// Check duration for each phase
positionExtrema := ruckig._profiles[0].positionExtrema();
AssertEquals_LREAL(8.0, positionExtrema.Tmax, 1E-9, message:='Profile[0] Tmax incorrect');
AssertEquals_LREAL(3112.370485074103, positionExtrema.Maximum, 1E-9, message:='Profile[0] maximum incorrect');
AssertEquals_LREAL(0.0, positionExtrema.Tmin, 1E-9, message:='Profile[0] Tmin incorrect');
AssertEquals_LREAL(78.42679297249512, positionExtrema.Minimum, 1E-9, message:='Profile[0] minimum incorrect');

positionExtrema := ruckig._profiles[1].positionExtrema();
AssertEquals_LREAL(0.2183891025126522, positionExtrema.Tmax, 1E-9, message:='Profile[1] Tmax incorrect');
AssertEquals_LREAL(46.54452205781156, positionExtrema.Maximum, 1E-9, message:='Profile[1] maximum incorrect');
AssertEquals_LREAL(8.0, positionExtrema.Tmin, 1E-9, message:='Profile[1] Tmin incorrect');
AssertEquals_LREAL(-9787.213398023361, positionExtrema.Minimum, 1E-9, message:='Profile[1] minimum incorrect');

positionExtrema := ruckig._profiles[2].positionExtrema();
AssertEquals_LREAL(0.0494303119629617, positionExtrema.Tmax, 1E-9, message:='Profile[2] Tmax incorrect');
AssertEquals_LREAL(31.710971182106867, positionExtrema.Maximum, 1E-9, message:='Profile[2] maximum incorrect');
AssertEquals_LREAL(8.0, positionExtrema.Tmin, 1E-9, message:='Profile[2] Tmin incorrect');
AssertEquals_LREAL(-8022.928301920572, positionExtrema.Minimum, 1E-9, message:='Profile[2] minimum incorrect');
   

TEST_FINISHED();
END_METHOD

METHOD Test_Trajectory_VelIntrf_HasMinDuration_HasTargetVelocity_HasTargetAcceleration_22
VAR_INST
  ruckig : Struckig.Ruckig(0.001, 3) := (
  
    ControlInterface := ControlInterfaceType.Velocity,
    Synchronization := SynchronizationType.TimeSync,
    MinDuration := 2.0,
    MaxVelocity := [ 2000.0, 2000.0, 2000.0 ],
    MaxAcceleration := [ 20000.0, 20000.0, 20000.0 ],
    MaxJerk := [ 800000.0, 800000.0, 800000.0 ],
    CurrentPosition := [ -79.7347950117767, 19.391476793099315, 7.245161501695378 ],
    CurrentVelocity := [ 143.04128173279923, -597.5124545779606, -118.71564531017145 ],
    CurrentAcceleration := [ 5642.529309782371, -4265.609648746094, 4828.540937996317 ],
    TargetPosition := [ -68.4590507631062, -68.46147249712232, -71.29488743466081 ],
    TargetVelocity := [ -770.5297588001531, -967.3934412952574, 417.4312367444536 ],
    TargetAcceleration := [ -41.66111920833407, 935.4765738277545, -963.8609114010426 ]
  );
  
  positionExtrema : Struckig.PositionExtremaDesc;
END_VAR
TEST('Trajectory_VelIntrf_HasMinDuration_HasTargetVelocity_HasTargetAcceleration_22');

ruckig();

// Check total duration of profiles
AssertEquals_LREAL(Expected := 2.0, Actual := ruckig.Duration, DELTA := 1E-8, Message := 'Duration incorrect');

// Check minimum duration
AssertEquals_LREAL(Expected := ruckig.MinDuration, Actual := ruckig.Duration, DELTA := 1E-8, Message := 'Minimum duration not equals duration');

// Check duration for each phase
positionExtrema := ruckig._profiles[0].positionExtrema();
AssertEquals_LREAL(0.007638802536377481, positionExtrema.Tmax, 1E-9, message:='Profile[0] Tmax incorrect');
AssertEquals_LREAL(-78.53693764605154, positionExtrema.Maximum, 1E-9, message:='Profile[0] maximum incorrect');
AssertEquals_LREAL(2.0, positionExtrema.Tmin, 1E-9, message:='Profile[0] Tmin incorrect');
AssertEquals_LREAL(-684.0560377921786, positionExtrema.Minimum, 1E-9, message:='Profile[0] minimum incorrect');

positionExtrema := ruckig._profiles[1].positionExtrema();
AssertEquals_LREAL(0.0, positionExtrema.Tmax, 1E-9, message:='Profile[1] Tmax incorrect');
AssertEquals_LREAL(19.391476793099315, positionExtrema.Maximum, 1E-9, message:='Profile[1] maximum incorrect');
AssertEquals_LREAL(2.0, positionExtrema.Tmin, 1E-9, message:='Profile[1] Tmin incorrect');
AssertEquals_LREAL(-3142.7217669332654, positionExtrema.Minimum, 1E-9, message:='Profile[1] minimum incorrect');

positionExtrema := ruckig._profiles[2].positionExtrema();
AssertEquals_LREAL(2.0, positionExtrema.Tmax, 1E-9, message:='Profile[2] Tmax incorrect');
AssertEquals_LREAL(2071.1384078495203, positionExtrema.Maximum, 1E-9, message:='Profile[2] maximum incorrect');
AssertEquals_LREAL(0.02502787930237134, positionExtrema.Tmin, 1E-9, message:='Profile[2] Tmin incorrect');
AssertEquals_LREAL(5.768456383094455, positionExtrema.Minimum, 1E-9, message:='Profile[2] minimum incorrect');
   

TEST_FINISHED();
END_METHOD

METHOD Test_Trajectory_VelIntrf_HasMinDuration_HasTargetVelocity_HasTargetAcceleration_23
VAR_INST
  ruckig : Struckig.Ruckig(0.001, 3) := (
  
    ControlInterface := ControlInterfaceType.Velocity,
    Synchronization := SynchronizationType.TimeSync,
    MinDuration := 4.0,
    MaxVelocity := [ 2000.0, 2000.0, 2000.0 ],
    MaxAcceleration := [ 20000.0, 20000.0, 20000.0 ],
    MaxJerk := [ 800000.0, 800000.0, 800000.0 ],
    CurrentPosition := [ 61.37396011937787, 91.70380359961769, -8.257039659155268 ],
    CurrentVelocity := [ -246.00859628849685, -467.85176399454747, -618.5921990326065 ],
    CurrentAcceleration := [ -4298.249657421169, 4989.7430906178615, -9033.185410088885 ],
    TargetPosition := [ -63.08099775805782, -90.41352080290159, -99.37485926962239 ],
    TargetVelocity := [ -239.3077646725386, 919.245352779569, -397.28894892304845 ],
    TargetAcceleration := [ -291.4115348913673, 23.504752198523192, -795.5915465895694 ]
  );
  
  positionExtrema : Struckig.PositionExtremaDesc;
END_VAR
TEST('Trajectory_VelIntrf_HasMinDuration_HasTargetVelocity_HasTargetAcceleration_23');

ruckig();

// Check total duration of profiles
AssertEquals_LREAL(Expected := 4.0, Actual := ruckig.Duration, DELTA := 1E-8, Message := 'Duration incorrect');

// Check minimum duration
AssertEquals_LREAL(Expected := ruckig.MinDuration, Actual := ruckig.Duration, DELTA := 1E-8, Message := 'Minimum duration not equals duration');

// Check duration for each phase
positionExtrema := ruckig._profiles[0].positionExtrema();
AssertEquals_LREAL(0.0, positionExtrema.Tmax, 1E-9, message:='Profile[0] Tmax incorrect');
AssertEquals_LREAL(61.37396011937787, positionExtrema.Maximum, 1E-9, message:='Profile[0] maximum incorrect');
AssertEquals_LREAL(4.0, positionExtrema.Tmin, 1E-9, message:='Profile[0] Tmin incorrect');
AssertEquals_LREAL(-932.2714554581783, positionExtrema.Minimum, 1E-9, message:='Profile[0] minimum incorrect');

positionExtrema := ruckig._profiles[1].positionExtrema();
AssertEquals_LREAL(4.0, positionExtrema.Tmax, 1E-9, message:='Profile[1] Tmax incorrect');
AssertEquals_LREAL(3356.191464991089, positionExtrema.Maximum, 1E-9, message:='Profile[1] maximum incorrect');
AssertEquals_LREAL(0.10412338784096734, positionExtrema.Tmin, 1E-9, message:='Profile[1] Tmin incorrect');
AssertEquals_LREAL(68.24379604148844, positionExtrema.Minimum, 1E-9, message:='Profile[1] minimum incorrect');

positionExtrema := ruckig._profiles[2].positionExtrema();
AssertEquals_LREAL(0.0, positionExtrema.Tmax, 1E-9, message:='Profile[2] Tmax incorrect');
AssertEquals_LREAL(-8.257039659155268, positionExtrema.Maximum, 1E-9, message:='Profile[2] maximum incorrect');
AssertEquals_LREAL(4.0, positionExtrema.Tmin, 1E-9, message:='Profile[2] Tmin incorrect');
AssertEquals_LREAL(-2142.4383401030323, positionExtrema.Minimum, 1E-9, message:='Profile[2] minimum incorrect');
   

TEST_FINISHED();
END_METHOD

METHOD Test_Trajectory_VelIntrf_HasMinDuration_HasTargetVelocity_HasTargetAcceleration_25
VAR_INST
  ruckig : Struckig.Ruckig(0.001, 3) := (
  
    ControlInterface := ControlInterfaceType.Velocity,
    Synchronization := SynchronizationType.TimeSync,
    MinDuration := 5.0,
    MaxVelocity := [ 2000.0, 2000.0, 2000.0 ],
    MaxAcceleration := [ 20000.0, 20000.0, 20000.0 ],
    MaxJerk := [ 800000.0, 800000.0, 800000.0 ],
    CurrentPosition := [ 99.27158709173054, 51.78630599017913, -82.71240030046118 ],
    CurrentVelocity := [ 617.0096879713556, 556.3356400770322, 654.4714219366203 ],
    CurrentAcceleration := [ 574.9072883020708, 8161.605381343747, 7215.343607485673 ],
    TargetPosition := [ -75.73302485201327, -76.60258111111662, -93.84383456920497 ],
    TargetVelocity := [ -134.5020942775601, 636.5230467842334, -659.8475456020238 ],
    TargetAcceleration := [ -262.53891173287866, -851.053910299499, -307.5361794862756 ]
  );
  
  positionExtrema : Struckig.PositionExtremaDesc;
END_VAR
TEST('Trajectory_VelIntrf_HasMinDuration_HasTargetVelocity_HasTargetAcceleration_25');

ruckig();

// Check total duration of profiles
AssertEquals_LREAL(Expected := 5.0, Actual := ruckig.Duration, DELTA := 1E-8, Message := 'Duration incorrect');

// Check minimum duration
AssertEquals_LREAL(Expected := ruckig.MinDuration, Actual := ruckig.Duration, DELTA := 1E-8, Message := 'Minimum duration not equals duration');

// Check duration for each phase
positionExtrema := ruckig._profiles[0].positionExtrema();
AssertEquals_LREAL(5.0, positionExtrema.Tmax, 1E-9, message:='Profile[0] Tmax incorrect');
AssertEquals_LREAL(2457.793957890017, positionExtrema.Maximum, 1E-9, message:='Profile[0] maximum incorrect');
AssertEquals_LREAL(0.0, positionExtrema.Tmin, 1E-9, message:='Profile[0] Tmin incorrect');
AssertEquals_LREAL(99.27158709173054, positionExtrema.Minimum, 1E-9, message:='Profile[0] minimum incorrect');

positionExtrema := ruckig._profiles[1].positionExtrema();
AssertEquals_LREAL(5.0, positionExtrema.Tmax, 1E-9, message:='Profile[1] Tmax incorrect');
AssertEquals_LREAL(12482.220923700503, positionExtrema.Maximum, 1E-9, message:='Profile[1] maximum incorrect');
AssertEquals_LREAL(0.0, positionExtrema.Tmin, 1E-9, message:='Profile[1] Tmin incorrect');
AssertEquals_LREAL(51.78630599017913, positionExtrema.Minimum, 1E-9, message:='Profile[1] minimum incorrect');

positionExtrema := ruckig._profiles[2].positionExtrema();
AssertEquals_LREAL(5.0, positionExtrema.Tmax, 1E-9, message:='Profile[2] Tmax incorrect');
AssertEquals_LREAL(457.83088712667626, positionExtrema.Maximum, 1E-9, message:='Profile[2] maximum incorrect');
AssertEquals_LREAL(0.0, positionExtrema.Tmin, 1E-9, message:='Profile[2] Tmin incorrect');
AssertEquals_LREAL(-82.71240030046118, positionExtrema.Minimum, 1E-9, message:='Profile[2] minimum incorrect');
   

TEST_FINISHED();
END_METHOD

METHOD Test_Trajectory_VelIntrf_HasMinDuration_HasTargetVelocity_HasTargetAcceleration_26
VAR_INST
  ruckig : Struckig.Ruckig(0.001, 3) := (
  
    ControlInterface := ControlInterfaceType.Velocity,
    Synchronization := SynchronizationType.TimeSync,
    MinDuration := 2.0,
    MaxVelocity := [ 2000.0, 2000.0, 2000.0 ],
    MaxAcceleration := [ 20000.0, 20000.0, 20000.0 ],
    MaxJerk := [ 800000.0, 800000.0, 800000.0 ],
    CurrentPosition := [ 47.83664173753348, -4.090200694219973, 75.62715399288581 ],
    CurrentVelocity := [ -412.71660212910535, -344.97977752529744, -662.3972561668236 ],
    CurrentAcceleration := [ 9700.323608694027, 4925.451680171778, 528.779511900253 ],
    TargetPosition := [ -26.350792724711255, -10.804969468053471, -80.84927076896919 ],
    TargetVelocity := [ -661.2515009925905, -544.0751045990595, 389.8586138148876 ],
    TargetAcceleration := [ -326.74185324603604, 477.02942558038353, -127.6960040536186 ]
  );
  
  positionExtrema : Struckig.PositionExtremaDesc;
END_VAR
TEST('Trajectory_VelIntrf_HasMinDuration_HasTargetVelocity_HasTargetAcceleration_26');

ruckig();

// Check total duration of profiles
AssertEquals_LREAL(Expected := 2.0, Actual := ruckig.Duration, DELTA := 1E-8, Message := 'Duration incorrect');

// Check minimum duration
AssertEquals_LREAL(Expected := ruckig.MinDuration, Actual := ruckig.Duration, DELTA := 1E-8, Message := 'Minimum duration not equals duration');

// Check duration for each phase
positionExtrema := ruckig._profiles[0].positionExtrema();
AssertEquals_LREAL(0.0, positionExtrema.Tmax, 1E-9, message:='Profile[0] Tmax incorrect');
AssertEquals_LREAL(47.83664173753348, positionExtrema.Maximum, 1E-9, message:='Profile[0] maximum incorrect');
AssertEquals_LREAL(2.0, positionExtrema.Tmin, 1E-9, message:='Profile[0] Tmin incorrect');
AssertEquals_LREAL(-965.6623915281051, positionExtrema.Minimum, 1E-9, message:='Profile[0] minimum incorrect');

positionExtrema := ruckig._profiles[1].positionExtrema();
AssertEquals_LREAL(0.0, positionExtrema.Tmax, 1E-9, message:='Profile[1] Tmax incorrect');
AssertEquals_LREAL(-4.090200694219973, positionExtrema.Maximum, 1E-9, message:='Profile[1] maximum incorrect');
AssertEquals_LREAL(2.0, positionExtrema.Tmin, 1E-9, message:='Profile[1] Tmin incorrect');
AssertEquals_LREAL(-877.5597601233831, positionExtrema.Minimum, 1E-9, message:='Profile[1] minimum incorrect');

positionExtrema := ruckig._profiles[2].positionExtrema();
AssertEquals_LREAL(0.0, positionExtrema.Tmax, 1E-9, message:='Profile[2] Tmax incorrect');
AssertEquals_LREAL(75.62715399288581, positionExtrema.Maximum, 1E-9, message:='Profile[2] maximum incorrect');
AssertEquals_LREAL(1.9991825530237812, positionExtrema.Tmin, 1E-9, message:='Profile[2] Tmin incorrect');
AssertEquals_LREAL(-196.96292798248453, positionExtrema.Minimum, 1E-9, message:='Profile[2] minimum incorrect');
   

TEST_FINISHED();
END_METHOD

METHOD Test_Trajectory_VelIntrf_HasMinDuration_HasTargetVelocity_HasTargetAcceleration_33
VAR_INST
  ruckig : Struckig.Ruckig(0.001, 3) := (
  
    ControlInterface := ControlInterfaceType.Velocity,
    Synchronization := SynchronizationType.TimeSync,
    MinDuration := 1.0,
    MaxVelocity := [ 2000.0, 2000.0, 2000.0 ],
    MaxAcceleration := [ 20000.0, 20000.0, 20000.0 ],
    MaxJerk := [ 800000.0, 800000.0, 800000.0 ],
    CurrentPosition := [ -49.2031444482373, -51.45640574706518, 70.88792157601674 ],
    CurrentVelocity := [ -496.32492650532754, -32.672137553484845, 433.6351152131574 ],
    CurrentAcceleration := [ 5796.767034802937, 149.52817879179565, 5479.773632181257 ],
    TargetPosition := [ -60.683308313785076, -77.36542095799315, 35.25281163323578 ],
    TargetVelocity := [ -239.87671609275264, 822.5237555037947, -341.77342454738846 ],
    TargetAcceleration := [ 442.7287565429956, -997.6913770242959, -816.4447449025389 ]
  );
  
  positionExtrema : Struckig.PositionExtremaDesc;
END_VAR
TEST('Trajectory_VelIntrf_HasMinDuration_HasTargetVelocity_HasTargetAcceleration_33');

ruckig();

// Check total duration of profiles
AssertEquals_LREAL(Expected := 1.0, Actual := ruckig.Duration, DELTA := 1E-8, Message := 'Duration incorrect');

// Check minimum duration
AssertEquals_LREAL(Expected := ruckig.MinDuration, Actual := ruckig.Duration, DELTA := 1E-8, Message := 'Minimum duration not equals duration');

// Check duration for each phase
positionExtrema := ruckig._profiles[0].positionExtrema();
AssertEquals_LREAL(0.0, positionExtrema.Tmax, 1E-9, message:='Profile[0] Tmax incorrect');
AssertEquals_LREAL(-49.2031444482373, positionExtrema.Maximum, 1E-9, message:='Profile[0] maximum incorrect');
AssertEquals_LREAL(1.0, positionExtrema.Tmin, 1E-9, message:='Profile[0] Tmin incorrect');
AssertEquals_LREAL(-407.7025966385173, positionExtrema.Minimum, 1E-9, message:='Profile[0] minimum incorrect');

positionExtrema := ruckig._profiles[1].positionExtrema();
AssertEquals_LREAL(1.0, positionExtrema.Tmax, 1E-9, message:='Profile[1] Tmax incorrect');
AssertEquals_LREAL(344.3868574234848, positionExtrema.Maximum, 1E-9, message:='Profile[1] maximum incorrect');
AssertEquals_LREAL(0.000885165723529272, positionExtrema.Tmin, 1E-9, message:='Profile[1] Tmin incorrect');
AssertEquals_LREAL(-51.485174951826146, positionExtrema.Minimum, 1E-9, message:='Profile[1] minimum incorrect');

positionExtrema := ruckig._profiles[2].positionExtrema();
AssertEquals_LREAL(0.9999795141123666, positionExtrema.Tmax, 1E-9, message:='Profile[2] Tmax incorrect');
AssertEquals_LREAL(129.085190687188, positionExtrema.Maximum, 1E-9, message:='Profile[2] maximum incorrect');
AssertEquals_LREAL(0.0, positionExtrema.Tmin, 1E-9, message:='Profile[2] Tmin incorrect');
AssertEquals_LREAL(70.88792157601674, positionExtrema.Minimum, 1E-9, message:='Profile[2] minimum incorrect');
   

TEST_FINISHED();
END_METHOD

METHOD Test_Trajectory_VelIntrf_HasMinDuration_HasTargetVelocity_HasTargetAcceleration_37
VAR_INST
  ruckig : Struckig.Ruckig(0.001, 3) := (
  
    ControlInterface := ControlInterfaceType.Velocity,
    Synchronization := SynchronizationType.TimeSync,
    MinDuration := 2.0,
    MaxVelocity := [ 2000.0, 2000.0, 2000.0 ],
    MaxAcceleration := [ 20000.0, 20000.0, 20000.0 ],
    MaxJerk := [ 800000.0, 800000.0, 800000.0 ],
    CurrentPosition := [ -12.004712599902348, 73.67282675877655, -52.349457595484836 ],
    CurrentVelocity := [ 292.20783385007076, -778.1307817801523, -64.33328614652999 ],
    CurrentAcceleration := [ 245.56834991156393, 4188.319168784961, -3762.4320312456057 ],
    TargetPosition := [ 82.49345668673473, 58.903290717842765, 34.45715254310531 ],
    TargetVelocity := [ -333.20598063149066, 685.2693740134762, 482.0796900333503 ],
    TargetAcceleration := [ 240.05556433564402, -666.6421184257438, -752.3384651343332 ]
  );
  
  positionExtrema : Struckig.PositionExtremaDesc;
END_VAR
TEST('Trajectory_VelIntrf_HasMinDuration_HasTargetVelocity_HasTargetAcceleration_37');

ruckig();

// Check total duration of profiles
AssertEquals_LREAL(Expected := 2.0, Actual := ruckig.Duration, DELTA := 1E-8, Message := 'Duration incorrect');

// Check minimum duration
AssertEquals_LREAL(Expected := ruckig.MinDuration, Actual := ruckig.Duration, DELTA := 1E-8, Message := 'Minimum duration not equals duration');

// Check duration for each phase
positionExtrema := ruckig._profiles[0].positionExtrema();
AssertEquals_LREAL(0.0006980853396357632, positionExtrema.Tmax, 1E-9, message:='Profile[0] Tmax incorrect');
AssertEquals_LREAL(-11.80071211848046, positionExtrema.Maximum, 1E-9, message:='Profile[0] maximum incorrect');
AssertEquals_LREAL(2.0, positionExtrema.Tmin, 1E-9, message:='Profile[0] Tmin incorrect');
AssertEquals_LREAL(-52.999031310760635, positionExtrema.Minimum, 1E-9, message:='Profile[0] minimum incorrect');

positionExtrema := ruckig._profiles[1].positionExtrema();
AssertEquals_LREAL(2.0, positionExtrema.Tmax, 1E-9, message:='Profile[1] Tmax incorrect');
AssertEquals_LREAL(1703.4819483796325, positionExtrema.Maximum, 1E-9, message:='Profile[1] maximum incorrect');
AssertEquals_LREAL(0.207432051719431, positionExtrema.Tmin, 1E-9, message:='Profile[1] Tmin incorrect');
AssertEquals_LREAL(-3.8974776087497673, positionExtrema.Minimum, 1E-9, message:='Profile[1] minimum incorrect');

positionExtrema := ruckig._profiles[2].positionExtrema();
AssertEquals_LREAL(2.0, positionExtrema.Tmax, 1E-9, message:='Profile[2] Tmax incorrect');
AssertEquals_LREAL(355.8717476818793, positionExtrema.Maximum, 1E-9, message:='Profile[2] maximum incorrect');
AssertEquals_LREAL(0.005051342367393055, positionExtrema.Tmin, 1E-9, message:='Profile[2] Tmin incorrect');
AssertEquals_LREAL(-52.70524288915402, positionExtrema.Minimum, 1E-9, message:='Profile[2] minimum incorrect');
   

TEST_FINISHED();
END_METHOD

METHOD Test_Trajectory_VelIntrf_HasMinDuration_HasTargetVelocity_HasTargetAcceleration_40
VAR_INST
  ruckig : Struckig.Ruckig(0.001, 3) := (
  
    ControlInterface := ControlInterfaceType.Velocity,
    Synchronization := SynchronizationType.TimeSync,
    MinDuration := 4.0,
    MaxVelocity := [ 2000.0, 2000.0, 2000.0 ],
    MaxAcceleration := [ 20000.0, 20000.0, 20000.0 ],
    MaxJerk := [ 800000.0, 800000.0, 800000.0 ],
    CurrentPosition := [ -76.42035041184897, -68.81061285502989, 60.15861595713818 ],
    CurrentVelocity := [ 424.8413928919874, 178.96533202855449, 765.6862190691088 ],
    CurrentAcceleration := [ 1338.04438518401, 3559.2301009959247, -1023.1564895528609 ],
    TargetPosition := [ -17.943807189703136, 56.757291906819944, -0.6309720814246589 ],
    TargetVelocity := [ -763.7685723303848, 641.2936977777251, -718.0886986858688 ],
    TargetAcceleration := [ 498.71648374610845, -601.18528422182, -73.467606210815 ]
  );
  
  positionExtrema : Struckig.PositionExtremaDesc;
END_VAR
TEST('Trajectory_VelIntrf_HasMinDuration_HasTargetVelocity_HasTargetAcceleration_40');

ruckig();

// Check total duration of profiles
AssertEquals_LREAL(Expected := 4.0, Actual := ruckig.Duration, DELTA := 1E-8, Message := 'Duration incorrect');

// Check minimum duration
AssertEquals_LREAL(Expected := ruckig.MinDuration, Actual := ruckig.Duration, DELTA := 1E-8, Message := 'Minimum duration not equals duration');

// Check duration for each phase
positionExtrema := ruckig._profiles[0].positionExtrema();
AssertEquals_LREAL(0.0020446425392176273, positionExtrema.Tmax, 1E-9, message:='Profile[0] Tmax incorrect');
AssertEquals_LREAL(-75.5500444389785, positionExtrema.Maximum, 1E-9, message:='Profile[0] maximum incorrect');
AssertEquals_LREAL(4.0, positionExtrema.Tmin, 1E-9, message:='Profile[0] Tmin incorrect');
AssertEquals_LREAL(-751.7240555499565, positionExtrema.Minimum, 1E-9, message:='Profile[0] minimum incorrect');

positionExtrema := ruckig._profiles[1].positionExtrema();
AssertEquals_LREAL(4.0, positionExtrema.Tmax, 1E-9, message:='Profile[1] Tmax incorrect');
AssertEquals_LREAL(5988.6562563663865, positionExtrema.Maximum, 1E-9, message:='Profile[1] maximum incorrect');
AssertEquals_LREAL(0.0, positionExtrema.Tmin, 1E-9, message:='Profile[1] Tmin incorrect');
AssertEquals_LREAL(-68.81061285502989, positionExtrema.Minimum, 1E-9, message:='Profile[1] minimum incorrect');

positionExtrema := ruckig._profiles[2].positionExtrema();
AssertEquals_LREAL(0.897558808059484, positionExtrema.Tmax, 1E-9, message:='Profile[2] Tmax incorrect');
AssertEquals_LREAL(380.9463968009695, positionExtrema.Maximum, 1E-9, message:='Profile[2] maximum incorrect');
AssertEquals_LREAL(4.0, positionExtrema.Tmin, 1E-9, message:='Profile[2] Tmin incorrect');
AssertEquals_LREAL(-1230.5349501304436, positionExtrema.Minimum, 1E-9, message:='Profile[2] minimum incorrect');
   

TEST_FINISHED();
END_METHOD

METHOD Test_Trajectory_VelIntrf_HasMinDuration_HasTargetVelocity_HasTargetAcceleration_9
VAR_INST
  ruckig : Struckig.Ruckig(0.001, 3) := (
  
    ControlInterface := ControlInterfaceType.Velocity,
    Synchronization := SynchronizationType.TimeSync,
    MinDuration := 7.0,
    MaxVelocity := [ 2000.0, 2000.0, 2000.0 ],
    MaxAcceleration := [ 20000.0, 20000.0, 20000.0 ],
    MaxJerk := [ 800000.0, 800000.0, 800000.0 ],
    CurrentPosition := [ 65.33675034249944, 20.471874067999465, 17.7936900678952 ],
    CurrentVelocity := [ 251.51375561632767, -883.355945316876, 592.220566480973 ],
    CurrentAcceleration := [ 9181.774579926536, -9976.3302467699, 2745.115542495065 ],
    TargetPosition := [ -63.4605755257718, 16.3093879856457, -25.6649619333392 ],
    TargetVelocity := [ 614.4494968030804, -34.17434532431503, 533.9879492839282 ],
    TargetAcceleration := [ -792.1476751145624, 673.4644110073796, -240.28714730173158 ]
  );
  
  positionExtrema : Struckig.PositionExtremaDesc;
END_VAR
TEST('Trajectory_VelIntrf_HasMinDuration_HasTargetVelocity_HasTargetAcceleration_9');

ruckig();

// Check total duration of profiles
AssertEquals_LREAL(Expected := 7.0, Actual := ruckig.Duration, DELTA := 1E-8, Message := 'Duration incorrect');

// Check minimum duration
AssertEquals_LREAL(Expected := ruckig.MinDuration, Actual := ruckig.Duration, DELTA := 1E-8, Message := 'Minimum duration not equals duration');

// Check duration for each phase
positionExtrema := ruckig._profiles[0].positionExtrema();
AssertEquals_LREAL(7.0, positionExtrema.Tmax, 1E-9, message:='Profile[0] Tmax incorrect');
AssertEquals_LREAL(21441.07705236427, positionExtrema.Maximum, 1E-9, message:='Profile[0] maximum incorrect');
AssertEquals_LREAL(0.0, positionExtrema.Tmin, 1E-9, message:='Profile[0] Tmin incorrect');
AssertEquals_LREAL(65.33675034249944, positionExtrema.Minimum, 1E-9, message:='Profile[0] minimum incorrect');

positionExtrema := ruckig._profiles[1].positionExtrema();
AssertEquals_LREAL(0.0, positionExtrema.Tmax, 1E-9, message:='Profile[1] Tmax incorrect');
AssertEquals_LREAL(20.471874067999465, positionExtrema.Maximum, 1E-9, message:='Profile[1] maximum incorrect');
AssertEquals_LREAL(7.0, positionExtrema.Tmin, 1E-9, message:='Profile[1] Tmin incorrect');
AssertEquals_LREAL(-15783.474903608412, positionExtrema.Minimum, 1E-9, message:='Profile[1] minimum incorrect');

positionExtrema := ruckig._profiles[2].positionExtrema();
AssertEquals_LREAL(7.0, positionExtrema.Tmax, 1E-9, message:='Profile[2] Tmax incorrect');
AssertEquals_LREAL(9053.9566289456, positionExtrema.Maximum, 1E-9, message:='Profile[2] maximum incorrect');
AssertEquals_LREAL(0.0, positionExtrema.Tmin, 1E-9, message:='Profile[2] Tmin incorrect');
AssertEquals_LREAL(17.7936900678952, positionExtrema.Minimum, 1E-9, message:='Profile[2] minimum incorrect');
   

TEST_FINISHED();
END_METHOD

END_FUNCTION_BLOCK

// ---- POUs/MinDurationTest.TcPOU
FUNCTION_BLOCK MinDurationTest EXTENDS TcUnit.FB_TestSuite

Test_Trajectory_HasMinDuration_HasTargetAcceleration_1();
Test_Trajectory_HasMinDuration_HasTargetAcceleration_2();
Test_Trajectory_HasMinDuration_HasTargetAcceleration_3();
Test_Trajectory_HasMinDuration_HasTargetAcceleration_4();
Test_Trajectory_HasMinDuration_HasTargetVelocity_5();
Test_Trajectory_HasMinDuration_HasTargetAcceleration_6();
Test_Trajectory_HasMinDuration_7();
Test_Trajectory_HasMinDuration_8();
Test_Trajectory_HasMinDuration_HasTargetVelocity_9();
Test_Trajectory_HasMinDuration_HasTargetVelocity_HasTargetAcceleration_10();
Test_Trajectory_HasMinDuration_HasTargetAcceleration_11();
Test_Trajectory_HasMinDuration_HasTargetVelocity_HasTargetAcceleration_12();
Test_Trajectory_HasMinDuration_13();
Test_Trajectory_HasMinDuration_14();
Test_Trajectory_HasMinDuration_HasTargetVelocity_HasTargetAcceleration_15();
Test_Trajectory_HasMinDuration_HasTargetVelocity_16();
Test_Trajectory_HasMinDuration_HasTargetAcceleration_17();
Test_Trajectory_HasMinDuration_HasTargetVelocity_HasTargetAcceleration_18();
Test_Trajectory_HasMinDuration_19();
Test_Trajectory_HasMinDuration_HasTargetVelocity_HasTargetAcceleration_20();

METHOD Test_Trajectory_HasMinDuration_13
VAR_INST
  ruckig : Struckig.Ruckig(0.001, 3) := (
  
    Synchronization := SynchronizationType.TimeSync,
    MinDuration := 8.0,
    MaxVelocity := [ 2000.0, 2000.0, 2000.0 ],
    MaxAcceleration := [ 20000.0, 20000.0, 20000.0 ],
    MaxJerk := [ 800000.0, 800000.0, 800000.0 ],
    CurrentPosition := [ 1.1694773064989192, -79.79875434933777, -86.29153082024368 ],
    CurrentVelocity := [ 876.2379533240828, 909.0293542700074, 204.90724883608482 ],
    CurrentAcceleration := [ -68.09095586171134, 4894.443101566274, 4257.694972396241 ],
    TargetPosition := [ -34.92331212819428, 11.554557728133503, 4.460284190197925 ],
    TargetVelocity := [ 0.0, 0.0, 0.0 ],
    TargetAcceleration := [ 0.0, 0.0, 0.0 ]
  );
  
  positionExtrema : Struckig.PositionExtremaDesc;
END_VAR
TEST('Trajectory_HasMinDuration_13');

ruckig();

// Check total duration of profiles
AssertEquals_LREAL(Expected := 8.0, Actual := ruckig.Duration, DELTA := 1E-8, Message := 'Duration incorrect');

// Check minimum duration
AssertEquals_LREAL(Expected := 8.0, Actual := ruckig.Duration, DELTA := 1E-8, Message := 'Duration incorrect');

// Check duration for each phase
positionExtrema := ruckig._profiles[0].positionExtrema();
AssertEquals_LREAL(0.06457933411638962, positionExtrema.Tmax, 1E-9, message:='Profile[0] Tmax incorrect');
AssertEquals_LREAL(31.162316883962312, positionExtrema.Maximum, 1E-9, message:='Profile[0] maximum incorrect');
AssertEquals_LREAL(7.999999999999999, positionExtrema.Tmin, 1E-9, message:='Profile[0] Tmin incorrect');
AssertEquals_LREAL(-34.92331212819428, positionExtrema.Minimum, 1E-9, message:='Profile[0] minimum incorrect');

positionExtrema := ruckig._profiles[1].positionExtrema();
AssertEquals_LREAL(8.0, positionExtrema.Tmax, 1E-9, message:='Profile[1] Tmax incorrect');
AssertEquals_LREAL(11.554557728133503, positionExtrema.Maximum, 1E-9, message:='Profile[1] maximum incorrect');
AssertEquals_LREAL(0.0, positionExtrema.Tmin, 1E-9, message:='Profile[1] Tmin incorrect');
AssertEquals_LREAL(-79.79875434933777, positionExtrema.Minimum, 1E-9, message:='Profile[1] minimum incorrect');

positionExtrema := ruckig._profiles[2].positionExtrema();
AssertEquals_LREAL(8.0, positionExtrema.Tmax, 1E-9, message:='Profile[2] Tmax incorrect');
AssertEquals_LREAL(4.460284190197925, positionExtrema.Maximum, 1E-9, message:='Profile[2] maximum incorrect');
AssertEquals_LREAL(0.0, positionExtrema.Tmin, 1E-9, message:='Profile[2] Tmin incorrect');
AssertEquals_LREAL(-86.29153082024368, positionExtrema.Minimum, 1E-9, message:='Profile[2] minimum incorrect');
   

TEST_FINISHED();
END_METHOD

METHOD Test_Trajectory_HasMinDuration_14
VAR_INST
  ruckig : Struckig.Ruckig(0.001, 3) := (
  
    Synchronization := SynchronizationType.TimeSync,
    MinDuration := 7.0,
    MaxVelocity := [ 2000.0, 2000.0, 2000.0 ],
    MaxAcceleration := [ 20000.0, 20000.0, 20000.0 ],
    MaxJerk := [ 800000.0, 800000.0, 800000.0 ],
    CurrentPosition := [ 9.590430768397383, 39.54262361303532, 47.91880435556814 ],
    CurrentVelocity := [ -279.73110233883074, -397.2798941946028, -792.783818655297 ],
    CurrentAcceleration := [ 9419.249088701486, -5244.89074121808, -9282.308244489752 ],
    TargetPosition := [ 70.18041902211951, 76.40810294125586, -12.064967166259137 ],
    TargetVelocity := [ 0.0, 0.0, 0.0 ],
    TargetAcceleration := [ 0.0, 0.0, 0.0 ]
  );
  
  positionExtrema : Struckig.PositionExtremaDesc;
END_VAR
TEST('Trajectory_HasMinDuration_14');

ruckig();

// Check total duration of profiles
AssertEquals_LREAL(Expected := 7.0, Actual := ruckig.Duration, DELTA := 1E-8, Message := 'Duration incorrect');

// Check minimum duration
AssertEquals_LREAL(Expected := 7.0, Actual := ruckig.Duration, DELTA := 1E-8, Message := 'Duration incorrect');

// Check duration for each phase
positionExtrema := ruckig._profiles[0].positionExtrema();
AssertEquals_LREAL(7.0, positionExtrema.Tmax, 1E-9, message:='Profile[0] Tmax incorrect');
AssertEquals_LREAL(70.18041902211951, positionExtrema.Maximum, 1E-9, message:='Profile[0] maximum incorrect');
AssertEquals_LREAL(0.024939596648417404, positionExtrema.Tmin, 1E-9, message:='Profile[0] Tmin incorrect');
AssertEquals_LREAL(6.5259576965994945, positionExtrema.Minimum, 1E-9, message:='Profile[0] minimum incorrect');

positionExtrema := ruckig._profiles[1].positionExtrema();
AssertEquals_LREAL(6.999999999999999, positionExtrema.Tmax, 1E-9, message:='Profile[1] Tmax incorrect');
AssertEquals_LREAL(76.40810294125586, positionExtrema.Maximum, 1E-9, message:='Profile[1] maximum incorrect');
AssertEquals_LREAL(0.0482688279337284, positionExtrema.Tmin, 1E-9, message:='Profile[1] Tmin incorrect');
AssertEquals_LREAL(27.490923337843135, positionExtrema.Minimum, 1E-9, message:='Profile[1] minimum incorrect');

positionExtrema := ruckig._profiles[2].positionExtrema();
AssertEquals_LREAL(0.0, positionExtrema.Tmax, 1E-9, message:='Profile[2] Tmax incorrect');
AssertEquals_LREAL(47.91880435556814, positionExtrema.Maximum, 1E-9, message:='Profile[2] maximum incorrect');
AssertEquals_LREAL(7.0, positionExtrema.Tmin, 1E-9, message:='Profile[2] Tmin incorrect');
AssertEquals_LREAL(-12.064967166259137, positionExtrema.Minimum, 1E-9, message:='Profile[2] minimum incorrect');
   

TEST_FINISHED();
END_METHOD

METHOD Test_Trajectory_HasMinDuration_19
VAR_INST
  ruckig : Struckig.Ruckig(0.001, 3) := (
  
    Synchronization := SynchronizationType.TimeSync,
    MinDuration := 3.0,
    MaxVelocity := [ 2000.0, 2000.0, 2000.0 ],
    MaxAcceleration := [ 20000.0, 20000.0, 20000.0 ],
    MaxJerk := [ 800000.0, 800000.0, 800000.0 ],
    CurrentPosition := [ 19.6107174579693, -14.671676826720102, -83.4266917323848 ],
    CurrentVelocity := [ -926.4357934162077, 856.3688940409422, -76.05611387446447 ],
    CurrentAcceleration := [ 8950.685844022108, -6737.3624163819, 7093.876397069776 ],
    TargetPosition := [ 45.75525505687679, -17.630601082354573, 68.42483173219557 ],
    TargetVelocity := [ 0.0, 0.0, 0.0 ],
    TargetAcceleration := [ 0.0, 0.0, 0.0 ]
  );
  
  positionExtrema : Struckig.PositionExtremaDesc;
END_VAR
TEST('Trajectory_HasMinDuration_19');

ruckig();

// Check total duration of profiles
AssertEquals_LREAL(Expected := 3.0, Actual := ruckig.Duration, DELTA := 1E-8, Message := 'Duration incorrect');

// Check minimum duration
AssertEquals_LREAL(Expected := 3.0, Actual := ruckig.Duration, DELTA := 1E-8, Message := 'Duration incorrect');

// Check duration for each phase
positionExtrema := ruckig._profiles[0].positionExtrema();
AssertEquals_LREAL(3.0, positionExtrema.Tmax, 1E-9, message:='Profile[0] Tmax incorrect');
AssertEquals_LREAL(45.75525505687679, positionExtrema.Maximum, 1E-9, message:='Profile[0] maximum incorrect');
AssertEquals_LREAL(0.05690150806828992, positionExtrema.Tmin, 1E-9, message:='Profile[0] Tmin incorrect');
AssertEquals_LREAL(-5.546975088681035, positionExtrema.Minimum, 1E-9, message:='Profile[0] minimum incorrect');

positionExtrema := ruckig._profiles[1].positionExtrema();
AssertEquals_LREAL(0.05654489225740592, positionExtrema.Tmax, 1E-9, message:='Profile[1] Tmax incorrect');
AssertEquals_LREAL(8.500086769282458, positionExtrema.Maximum, 1E-9, message:='Profile[1] maximum incorrect');
AssertEquals_LREAL(2.9999999999999996, positionExtrema.Tmin, 1E-9, message:='Profile[1] Tmin incorrect');
AssertEquals_LREAL(-17.630601082354573, positionExtrema.Minimum, 1E-9, message:='Profile[1] minimum incorrect');

positionExtrema := ruckig._profiles[2].positionExtrema();
AssertEquals_LREAL(3.0, positionExtrema.Tmax, 1E-9, message:='Profile[2] Tmax incorrect');
AssertEquals_LREAL(68.42483173219557, positionExtrema.Maximum, 1E-9, message:='Profile[2] maximum incorrect');
AssertEquals_LREAL(0.007991851854731072, positionExtrema.Tmin, 1E-9, message:='Profile[2] Tmin incorrect');
AssertEquals_LREAL(-83.74565322946518, positionExtrema.Minimum, 1E-9, message:='Profile[2] minimum incorrect');
   

TEST_FINISHED();
END_METHOD

METHOD Test_Trajectory_HasMinDuration_7
VAR_INST
  ruckig : Struckig.Ruckig(0.001, 3) := (
  
    Synchronization := SynchronizationType.TimeSync,
    MinDuration := 3.0,
    MaxVelocity := [ 2000.0, 2000.0, 2000.0 ],
    MaxAcceleration := [ 20000.0, 20000.0, 20000.0 ],
    MaxJerk := [ 800000.0, 800000.0, 800000.0 ],
    CurrentPosition := [ -29.448435809827217, 90.57043249467455, -42.4422398449114 ],
    CurrentVelocity := [ -441.1423852905707, 792.9273075694584, 308.64691156030153 ],
    CurrentAcceleration := [ -114.57718650638526, -7587.445490507809, 1437.7422990266587 ],
    TargetPosition := [ -44.03078989692402, 83.77708613438409, -82.0575436244257 ],
    TargetVelocity := [ 0.0, 0.0, 0.0 ],
    TargetAcceleration := [ 0.0, 0.0, 0.0 ]
  );
  
  positionExtrema : Struckig.PositionExtremaDesc;
END_VAR
TEST('Trajectory_HasMinDuration_7');

ruckig();

// Check total duration of profiles
AssertEquals_LREAL(Expected := 3.0, Actual := ruckig.Duration, DELTA := 1E-8, Message := 'Duration incorrect');

// Check minimum duration
AssertEquals_LREAL(Expected := 3.0, Actual := ruckig.Duration, DELTA := 1E-8, Message := 'Duration incorrect');

// Check duration for each phase
positionExtrema := ruckig._profiles[0].positionExtrema();
AssertEquals_LREAL(0.0, positionExtrema.Tmax, 1E-9, message:='Profile[0] Tmax incorrect');
AssertEquals_LREAL(-29.448435809827217, positionExtrema.Maximum, 1E-9, message:='Profile[0] maximum incorrect');
AssertEquals_LREAL(3.0, positionExtrema.Tmin, 1E-9, message:='Profile[0] Tmin incorrect');
AssertEquals_LREAL(-44.03078989692402, positionExtrema.Minimum, 1E-9, message:='Profile[0] minimum incorrect');

positionExtrema := ruckig._profiles[1].positionExtrema();
AssertEquals_LREAL(0.05266649608484671, positionExtrema.Tmax, 1E-9, message:='Profile[1] Tmax incorrect');
AssertEquals_LREAL(110.27502355296447, positionExtrema.Maximum, 1E-9, message:='Profile[1] maximum incorrect');
AssertEquals_LREAL(3.0, positionExtrema.Tmin, 1E-9, message:='Profile[1] Tmin incorrect');
AssertEquals_LREAL(83.77708613438409, positionExtrema.Minimum, 1E-9, message:='Profile[1] minimum incorrect');

positionExtrema := ruckig._profiles[2].positionExtrema();
AssertEquals_LREAL(0.03589522362162333, positionExtrema.Tmax, 1E-9, message:='Profile[2] Tmax incorrect');
AssertEquals_LREAL(-35.88360266407321, positionExtrema.Maximum, 1E-9, message:='Profile[2] maximum incorrect');
AssertEquals_LREAL(3.0000000000000004, positionExtrema.Tmin, 1E-9, message:='Profile[2] Tmin incorrect');
AssertEquals_LREAL(-82.0575436244257, positionExtrema.Minimum, 1E-9, message:='Profile[2] minimum incorrect');
   

TEST_FINISHED();
END_METHOD

METHOD Test_Trajectory_HasMinDuration_8
VAR_INST
  ruckig : Struckig.Ruckig(0.001, 3) := (
  
    Synchronization := SynchronizationType.TimeSync,
    MinDuration := 7.0,
    MaxVelocity := [ 2000.0, 2000.0, 2000.0 ],
    MaxAcceleration := [ 20000.0, 20000.0, 20000.0 ],
    MaxJerk := [ 800000.0, 800000.0, 800000.0 ],
    CurrentPosition := [ -99.24620189721642, 98.804478840699, -87.42756778236038 ],
    CurrentVelocity := [ -829.4036440965908, 623.2680808978928, 45.75080930558306 ],
    CurrentAcceleration := [ -7246.76941372717, 1502.5540766079612, -230.12493771912523 ],
    TargetPosition := [ -96.24866507944863, -68.29579645255217, 3.1547755930834427 ],
    TargetVelocity := [ 0.0, 0.0, 0.0 ],
    TargetAcceleration := [ 0.0, 0.0, 0.0 ]
  );
  
  positionExtrema : Struckig.PositionExtremaDesc;
END_VAR
TEST('Trajectory_HasMinDuration_8');

ruckig();

// Check total duration of profiles
AssertEquals_LREAL(Expected := 7.0, Actual := ruckig.Duration, DELTA := 1E-8, Message := 'Duration incorrect');

// Check minimum duration
AssertEquals_LREAL(Expected := 7.0, Actual := ruckig.Duration, DELTA := 1E-8, Message := 'Duration incorrect');

// Check duration for each phase
positionExtrema := ruckig._profiles[0].positionExtrema();
AssertEquals_LREAL(6.999999999999999, positionExtrema.Tmax, 1E-9, message:='Profile[0] Tmax incorrect');
AssertEquals_LREAL(-96.24866507944863, positionExtrema.Maximum, 1E-9, message:='Profile[0] maximum incorrect');
AssertEquals_LREAL(0.07365733450421347, positionExtrema.Tmin, 1E-9, message:='Profile[0] Tmin incorrect');
AssertEquals_LREAL(-136.26275842325944, positionExtrema.Minimum, 1E-9, message:='Profile[0] minimum incorrect');

positionExtrema := ruckig._profiles[1].positionExtrema();
AssertEquals_LREAL(0.05127223962572218, positionExtrema.Tmax, 1E-9, message:='Profile[1] Tmax incorrect');
AssertEquals_LREAL(117.33454096897361, positionExtrema.Maximum, 1E-9, message:='Profile[1] maximum incorrect');
AssertEquals_LREAL(7.000000000000001, positionExtrema.Tmin, 1E-9, message:='Profile[1] Tmin incorrect');
AssertEquals_LREAL(-68.29579645255217, positionExtrema.Minimum, 1E-9, message:='Profile[1] minimum incorrect');

positionExtrema := ruckig._profiles[2].positionExtrema();
AssertEquals_LREAL(7.000000000000001, positionExtrema.Tmax, 1E-9, message:='Profile[2] Tmax incorrect');
AssertEquals_LREAL(3.1547755930834427, positionExtrema.Maximum, 1E-9, message:='Profile[2] maximum incorrect');
AssertEquals_LREAL(0.0, positionExtrema.Tmin, 1E-9, message:='Profile[2] Tmin incorrect');
AssertEquals_LREAL(-87.42756778236038, positionExtrema.Minimum, 1E-9, message:='Profile[2] minimum incorrect');
   

TEST_FINISHED();
END_METHOD

METHOD Test_Trajectory_HasMinDuration_HasTargetAcceleration_1
VAR_INST
  ruckig : Struckig.Ruckig(0.001, 3) := (
    Synchronization := SynchronizationType.TimeSync,
    MinDuration := 8.0,
    MaxVelocity := [ 2000.0, 2000.0, 2000.0 ],
    MaxAcceleration := [ 20000.0, 20000.0, 20000.0 ],
    MaxJerk := [ 800000.0, 800000.0, 800000.0 ],
    CurrentPosition := [ -19.81606164381961, 13.781968848302611, 8.093103744301672 ],
    CurrentVelocity := [ 726.8874662814426, 243.71684078988915, 635.9493654202183 ],
    CurrentAcceleration := [ 3652.605974217926, 644.8054101513426, -2503.0584587977 ],
    TargetPosition := [ -37.94747764035489, 31.097009748141545, 51.041074550360605 ],
    TargetVelocity := [ 0.0, 0.0, 0.0 ],
    TargetAcceleration := [ -885.392846257796, -430.70238502743985, -347.6934578997044 ]
  );
  
  positionExtrema : Struckig.PositionExtremaDesc;	
END_VAR
TEST('Trajectory_HasMinDuration_HasTargetAcceleration_1');

ruckig();

// Check total duration of profiles
AssertEquals_LREAL(Expected := 8.0, Actual := ruckig.Duration, DELTA := 1E-8, Message := 'Duration incorrect');

// Check minimum duration
AssertEquals_LREAL(Expected := 8.0, Actual := ruckig.Duration, DELTA := 1E-8, Message := 'Duration incorrect');

// Check duration for each phase
positionExtrema := ruckig._profiles[0].positionExtrema();
AssertEquals_LREAL(0.06287595543262448, positionExtrema.Tmax, 1E-9, message:='Profile[0] Tmax incorrect');
AssertEquals_LREAL(6.175884472766756, positionExtrema.Maximum, 1E-9, message:='Profile[0] maximum incorrect');
AssertEquals_LREAL(7.9977865178843555, positionExtrema.Tmin, 1E-9, message:='Profile[0] Tmin incorrect');
AssertEquals_LREAL(-37.94820063785038, positionExtrema.Minimum, 1E-9, message:='Profile[0] minimum incorrect');

positionExtrema := ruckig._profiles[1].positionExtrema();
AssertEquals_LREAL(7.999999999999999, positionExtrema.Tmax, 1E-9, message:='Profile[1] Tmax incorrect');
AssertEquals_LREAL(31.097009748141545, positionExtrema.Maximum, 1E-9, message:='Profile[1] maximum incorrect');
AssertEquals_LREAL(0.0, positionExtrema.Tmin, 1E-9, message:='Profile[1] Tmin incorrect');
AssertEquals_LREAL(13.781968848302611, positionExtrema.Minimum, 1E-9, message:='Profile[1] minimum incorrect');

positionExtrema := ruckig._profiles[2].positionExtrema();
AssertEquals_LREAL(8.0, positionExtrema.Tmax, 1E-9, message:='Profile[2] Tmax incorrect');
AssertEquals_LREAL(51.041074550360605, positionExtrema.Maximum, 1E-9, message:='Profile[2] maximum incorrect');
AssertEquals_LREAL(0.0, positionExtrema.Tmin, 1E-9, message:='Profile[2] Tmin incorrect');
AssertEquals_LREAL(8.093103744301672, positionExtrema.Minimum, 1E-9, message:='Profile[2] minimum incorrect');
   

TEST_FINISHED();
END_METHOD

METHOD Test_Trajectory_HasMinDuration_HasTargetAcceleration_11
VAR_INST
  ruckig : Struckig.Ruckig(0.001, 3) := (
  
    Synchronization := SynchronizationType.TimeSync,
    MinDuration := 1.0,
    MaxVelocity := [ 2000.0, 2000.0, 2000.0 ],
    MaxAcceleration := [ 20000.0, 20000.0, 20000.0 ],
    MaxJerk := [ 800000.0, 800000.0, 800000.0 ],
    CurrentPosition := [ -7.070165280610553, -80.38372522590178, -46.89812209342119 ],
    CurrentVelocity := [ 839.4919555565891, -203.32957691775698, 521.9568411481566 ],
    CurrentAcceleration := [ 3262.1046041862974, -1428.6156287598897, 5033.848829385297 ],
    TargetPosition := [ 39.58959333241566, -77.56627414027115, -4.797228333391573 ],
    TargetVelocity := [ 0.0, 0.0, 0.0 ],
    TargetAcceleration := [ -610.5754269308525, -729.7372379589295, -407.1344521857434 ]
  );
  
  positionExtrema : Struckig.PositionExtremaDesc;
END_VAR
TEST('Trajectory_HasMinDuration_HasTargetAcceleration_11');

ruckig();

// Check total duration of profiles
AssertEquals_LREAL(Expected := 1.0, Actual := ruckig.Duration, DELTA := 1E-8, Message := 'Duration incorrect');

// Check minimum duration
AssertEquals_LREAL(Expected := 1.0, Actual := ruckig.Duration, DELTA := 1E-8, Message := 'Duration incorrect');

// Check duration for each phase
positionExtrema := ruckig._profiles[0].positionExtrema();
AssertEquals_LREAL(1.0, positionExtrema.Tmax, 1E-9, message:='Profile[0] Tmax incorrect');
AssertEquals_LREAL(39.58959333241566, positionExtrema.Maximum, 1E-9, message:='Profile[0] maximum incorrect');
AssertEquals_LREAL(0.0, positionExtrema.Tmin, 1E-9, message:='Profile[0] Tmin incorrect');
AssertEquals_LREAL(-7.070165280610553, positionExtrema.Minimum, 1E-9, message:='Profile[0] minimum incorrect');

positionExtrema := ruckig._profiles[1].positionExtrema();
AssertEquals_LREAL(1.0, positionExtrema.Tmax, 1E-9, message:='Profile[1] Tmax incorrect');
AssertEquals_LREAL(-77.56627414027115, positionExtrema.Maximum, 1E-9, message:='Profile[1] maximum incorrect');
AssertEquals_LREAL(0.030210863301643, positionExtrema.Tmin, 1E-9, message:='Profile[1] Tmin incorrect');
AssertEquals_LREAL(-83.98327189159232, positionExtrema.Minimum, 1E-9, message:='Profile[1] minimum incorrect');

positionExtrema := ruckig._profiles[2].positionExtrema();
AssertEquals_LREAL(1.0000000000000002, positionExtrema.Tmax, 1E-9, message:='Profile[2] Tmax incorrect');
AssertEquals_LREAL(-4.797228333391573, positionExtrema.Maximum, 1E-9, message:='Profile[2] maximum incorrect');
AssertEquals_LREAL(0.0, positionExtrema.Tmin, 1E-9, message:='Profile[2] Tmin incorrect');
AssertEquals_LREAL(-46.89812209342119, positionExtrema.Minimum, 1E-9, message:='Profile[2] minimum incorrect');
   

TEST_FINISHED();
END_METHOD

METHOD Test_Trajectory_HasMinDuration_HasTargetAcceleration_17
VAR_INST
  ruckig : Struckig.Ruckig(0.001, 3) := (
  
    Synchronization := SynchronizationType.TimeSync,
    MinDuration := 10.0,
    MaxVelocity := [ 2000.0, 2000.0, 2000.0 ],
    MaxAcceleration := [ 20000.0, 20000.0, 20000.0 ],
    MaxJerk := [ 800000.0, 800000.0, 800000.0 ],
    CurrentPosition := [ 41.06103962416182, -31.80504488955978, 63.99589133347962 ],
    CurrentVelocity := [ -749.439069786537, -605.1709178805476, -675.8190572055869 ],
    CurrentAcceleration := [ 4505.221832985957, 2158.0191432223, -7626.549080643861 ],
    TargetPosition := [ -49.277633620043005, -77.94196192090983, 7.643571349353522 ],
    TargetVelocity := [ 0.0, 0.0, 0.0 ],
    TargetAcceleration := [ -613.4884636354268, -619.351295536964, -177.16987102998473 ]
  );
  
  positionExtrema : Struckig.PositionExtremaDesc;
END_VAR
TEST('Trajectory_HasMinDuration_HasTargetAcceleration_17');

ruckig();

// Check total duration of profiles
AssertEquals_LREAL(Expected := 10.0, Actual := ruckig.Duration, DELTA := 1E-8, Message := 'Duration incorrect');

// Check minimum duration
AssertEquals_LREAL(Expected := 10.0, Actual := ruckig.Duration, DELTA := 1E-8, Message := 'Duration incorrect');

// Check duration for each phase
positionExtrema := ruckig._profiles[0].positionExtrema();
AssertEquals_LREAL(0.0, positionExtrema.Tmax, 1E-9, message:='Profile[0] Tmax incorrect');
AssertEquals_LREAL(41.06103962416182, positionExtrema.Maximum, 1E-9, message:='Profile[0] maximum incorrect');
AssertEquals_LREAL(9.998466278840914, positionExtrema.Tmin, 1E-9, message:='Profile[0] Tmin incorrect');
AssertEquals_LREAL(-49.27787413825579, positionExtrema.Minimum, 1E-9, message:='Profile[0] minimum incorrect');

positionExtrema := ruckig._profiles[1].positionExtrema();
AssertEquals_LREAL(0.0, positionExtrema.Tmax, 1E-9, message:='Profile[1] Tmax incorrect');
AssertEquals_LREAL(-31.80504488955978, positionExtrema.Maximum, 1E-9, message:='Profile[1] maximum incorrect');
AssertEquals_LREAL(9.99845162176116, positionExtrema.Tmin, 1E-9, message:='Profile[1] Tmin incorrect');
AssertEquals_LREAL(-77.94220940080136, positionExtrema.Minimum, 1E-9, message:='Profile[1] minimum incorrect');

positionExtrema := ruckig._profiles[2].positionExtrema();
AssertEquals_LREAL(0.0, positionExtrema.Tmax, 1E-9, message:='Profile[2] Tmax incorrect');
AssertEquals_LREAL(63.99589133347962, positionExtrema.Maximum, 1E-9, message:='Profile[2] maximum incorrect');
AssertEquals_LREAL(9.999557075322427, positionExtrema.Tmin, 1E-9, message:='Profile[2] Tmin incorrect');
AssertEquals_LREAL(7.643565556420371, positionExtrema.Minimum, 1E-9, message:='Profile[2] minimum incorrect');
   

TEST_FINISHED();
END_METHOD

METHOD Test_Trajectory_HasMinDuration_HasTargetAcceleration_2
VAR_INST
  ruckig : Struckig.Ruckig(0.001, 3) := (
  
    Synchronization := SynchronizationType.TimeSync,
    MinDuration := 9.0,
    MaxVelocity := [ 2000.0, 2000.0, 2000.0 ],
    MaxAcceleration := [ 20000.0, 20000.0, 20000.0 ],
    MaxJerk := [ 800000.0, 800000.0, 800000.0 ],
    CurrentPosition := [ 66.72445317186691, -7.406214437890085, 70.46458426730621 ],
    CurrentVelocity := [ 342.4260974225069, 430.1494125839465, -220.57495791564202 ],
    CurrentAcceleration := [ -4058.8697131936115, -937.4004804082579, -453.3153688510465 ],
    TargetPosition := [ 81.54050823089204, 50.65362401587811, 41.70097854809535 ],
    TargetVelocity := [ 0.0, 0.0, 0.0 ],
    TargetAcceleration := [ -58.178994858405304, 929.3098774625403, 47.05996186659536 ]
  );
  
  positionExtrema : Struckig.PositionExtremaDesc;
END_VAR
TEST('Trajectory_HasMinDuration_HasTargetAcceleration_2');

ruckig();

// Check total duration of profiles
AssertEquals_LREAL(Expected := 9.0, Actual := ruckig.Duration, DELTA := 1E-8, Message := 'Duration incorrect');

// Check minimum duration
AssertEquals_LREAL(Expected := ruckig.MinDuration, Actual := ruckig.Duration, DELTA := 1E-8, Message := 'Duration incorrect');

// Check duration for each phase
positionExtrema := ruckig._profiles[0].positionExtrema();
AssertEquals_LREAL(8.999999999999998, positionExtrema.Tmax, 1E-9, message:='Profile[0] Tmax incorrect');
AssertEquals_LREAL(81.54050823089204, positionExtrema.Maximum, 1E-9, message:='Profile[0] maximum incorrect');
AssertEquals_LREAL(0.0, positionExtrema.Tmin, 1E-9, message:='Profile[0] Tmin incorrect');
AssertEquals_LREAL(66.72445317186691, positionExtrema.Minimum, 1E-9, message:='Profile[0] minimum incorrect');

positionExtrema := ruckig._profiles[1].positionExtrema();
AssertEquals_LREAL(8.997676725306345, positionExtrema.Tmax, 1E-9, message:='Profile[1] Tmax incorrect');
AssertEquals_LREAL(50.65446002386552, positionExtrema.Maximum, 1E-9, message:='Profile[1] maximum incorrect');
AssertEquals_LREAL(0.0, positionExtrema.Tmin, 1E-9, message:='Profile[1] Tmin incorrect');
AssertEquals_LREAL(-7.406214437890085, positionExtrema.Minimum, 1E-9, message:='Profile[1] minimum incorrect');

positionExtrema := ruckig._profiles[2].positionExtrema();
AssertEquals_LREAL(0.0, positionExtrema.Tmax, 1E-9, message:='Profile[2] Tmax incorrect');
AssertEquals_LREAL(70.46458426730621, positionExtrema.Maximum, 1E-9, message:='Profile[2] maximum incorrect');
AssertEquals_LREAL(9.0, positionExtrema.Tmin, 1E-9, message:='Profile[2] Tmin incorrect');
AssertEquals_LREAL(41.70097854809503, positionExtrema.Minimum, 1E-9, message:='Profile[2] minimum incorrect');
   

TEST_FINISHED();
END_METHOD

METHOD Test_Trajectory_HasMinDuration_HasTargetAcceleration_3
VAR_INST
  ruckig : Struckig.Ruckig(0.001, 3) := (
  
    Synchronization := SynchronizationType.TimeSync,
    MinDuration := 7.0,
    MaxVelocity := [ 2000.0, 2000.0, 2000.0 ],
    MaxAcceleration := [ 20000.0, 20000.0, 20000.0 ],
    MaxJerk := [ 800000.0, 800000.0, 800000.0 ],
    CurrentPosition := [ 92.93281918195305, -37.057893567967405, -56.41888208246879 ],
    CurrentVelocity := [ 919.2036906054796, -544.1333420501469, 731.0755464554313 ],
    CurrentAcceleration := [ -7047.99292674085, 7580.284725007419, -3564.1022106007276 ],
    TargetPosition := [ -46.16949731931599, 10.423824279825439, 25.094577416282803 ],
    TargetVelocity := [ 0.0, 0.0, 0.0 ],
    TargetAcceleration := [ -597.0749810615916, 575.2171643962115, 815.8548576022943 ]
  );
  
  positionExtrema : Struckig.PositionExtremaDesc;
END_VAR
TEST('Trajectory_HasMinDuration_HasTargetAcceleration_3');

ruckig();

// Check total duration of profiles
AssertEquals_LREAL(Expected := 7.0, Actual := ruckig.Duration, DELTA := 1E-8, Message := 'Duration incorrect');

// Check minimum duration
AssertEquals_LREAL(Expected := 7.0, Actual := ruckig.Duration, DELTA := 1E-8, Message := 'Duration incorrect');

// Check duration for each phase
positionExtrema := ruckig._profiles[0].positionExtrema();
AssertEquals_LREAL(0.05717797410396826, positionExtrema.Tmax, 1E-9, message:='Profile[0] Tmax incorrect');
AssertEquals_LREAL(118.91548267627095, positionExtrema.Maximum, 1E-9, message:='Profile[0] maximum incorrect');
AssertEquals_LREAL(6.998507312547345, positionExtrema.Tmin, 1E-9, message:='Profile[0] Tmin incorrect');
AssertEquals_LREAL(-46.169719044685195, positionExtrema.Minimum, 1E-9, message:='Profile[0] minimum incorrect');

positionExtrema := ruckig._profiles[1].positionExtrema();
AssertEquals_LREAL(6.99856195708901, positionExtrema.Tmax, 1E-9, message:='Profile[1] Tmax incorrect');
AssertEquals_LREAL(10.424022534884019, positionExtrema.Maximum, 1E-9, message:='Profile[1] maximum incorrect');
AssertEquals_LREAL(0.0403879580291395, positionExtrema.Tmin, 1E-9, message:='Profile[1] Tmin incorrect');
AssertEquals_LREAL(-47.256877517684565, positionExtrema.Minimum, 1E-9, message:='Profile[1] minimum incorrect');

positionExtrema := ruckig._profiles[2].positionExtrema();
AssertEquals_LREAL(6.997960362855993, positionExtrema.Tmax, 1E-9, message:='Profile[2] Tmax incorrect');
AssertEquals_LREAL(25.095143091923283, positionExtrema.Maximum, 1E-9, message:='Profile[2] maximum incorrect');
AssertEquals_LREAL(0.0, positionExtrema.Tmin, 1E-9, message:='Profile[2] Tmin incorrect');
AssertEquals_LREAL(-56.41888208246879, positionExtrema.Minimum, 1E-9, message:='Profile[2] minimum incorrect');
   

TEST_FINISHED();
END_METHOD

METHOD Test_Trajectory_HasMinDuration_HasTargetAcceleration_4
VAR_INST
  ruckig : Struckig.Ruckig(0.001, 3) := (
  
    Synchronization := SynchronizationType.TimeSync,
    MinDuration := 3.0,
    MaxVelocity := [ 2000.0, 2000.0, 2000.0 ],
    MaxAcceleration := [ 20000.0, 20000.0, 20000.0 ],
    MaxJerk := [ 800000.0, 800000.0, 800000.0 ],
    CurrentPosition := [ -0.660339003647124, -95.83458227326918, -56.22509427236879 ],
    CurrentVelocity := [ -379.1557497186742, 437.2615639977953, 470.58690692947357 ],
    CurrentAcceleration := [ 7762.154315281241, -3727.206686180866, 7593.740905155453 ],
    TargetPosition := [ 84.07152685095582, 75.93155527258662, 84.6954649863176 ],
    TargetVelocity := [ 0.0, 0.0, 0.0 ],
    TargetAcceleration := [ -770.0559965976834, 741.3940743654641, -31.453470585175637 ]
  );
  
  positionExtrema : Struckig.PositionExtremaDesc;
END_VAR
TEST('Trajectory_HasMinDuration_HasTargetAcceleration_4');

ruckig();

// Check total duration of profiles
AssertEquals_LREAL(Expected := 3.0, Actual := ruckig.Duration, DELTA := 1E-8, Message := 'Duration incorrect');

// Check minimum duration
AssertEquals_LREAL(Expected := 3.0, Actual := ruckig.Duration, DELTA := 1E-8, Message := 'Duration incorrect');

// Check duration for each phase
positionExtrema := ruckig._profiles[0].positionExtrema();
AssertEquals_LREAL(2.9999999999999996, positionExtrema.Tmax, 1E-9, message:='Profile[0] Tmax incorrect');
AssertEquals_LREAL(84.07152685095582, positionExtrema.Maximum, 1E-9, message:='Profile[0] maximum incorrect');
AssertEquals_LREAL(0.028865029140955737, positionExtrema.Tmin, 1E-9, message:='Profile[0] Tmin incorrect');
AssertEquals_LREAL(-6.050680420215579, positionExtrema.Minimum, 1E-9, message:='Profile[0] minimum incorrect');

positionExtrema := ruckig._profiles[1].positionExtrema();
AssertEquals_LREAL(2.9981465148140867, positionExtrema.Tmax, 1E-9, message:='Profile[1] Tmax incorrect');
AssertEquals_LREAL(75.93197977102668, positionExtrema.Maximum, 1E-9, message:='Profile[1] maximum incorrect');
AssertEquals_LREAL(0.0, positionExtrema.Tmin, 1E-9, message:='Profile[1] Tmin incorrect');
AssertEquals_LREAL(-95.83458227326918, positionExtrema.Minimum, 1E-9, message:='Profile[1] minimum incorrect');

positionExtrema := ruckig._profiles[2].positionExtrema();
AssertEquals_LREAL(2.9999999999999987, positionExtrema.Tmax, 1E-9, message:='Profile[2] Tmax incorrect');
AssertEquals_LREAL(84.69546498631772, positionExtrema.Maximum, 1E-9, message:='Profile[2] maximum incorrect');
AssertEquals_LREAL(0.0, positionExtrema.Tmin, 1E-9, message:='Profile[2] Tmin incorrect');
AssertEquals_LREAL(-56.22509427236879, positionExtrema.Minimum, 1E-9, message:='Profile[2] minimum incorrect');
   

TEST_FINISHED();
END_METHOD

METHOD Test_Trajectory_HasMinDuration_HasTargetAcceleration_6
VAR_INST
  ruckig : Struckig.Ruckig(0.001, 3) := (
  
    Synchronization := SynchronizationType.TimeSync,
    MinDuration := 10.0,
    MaxVelocity := [ 2000.0, 2000.0, 2000.0 ],
    MaxAcceleration := [ 20000.0, 20000.0, 20000.0 ],
    MaxJerk := [ 800000.0, 800000.0, 800000.0 ],
    CurrentPosition := [ 73.95774355738217, 67.34262397589043, 23.586005113842518 ],
    CurrentVelocity := [ -698.8785963385769, -727.2426189740956, 561.2286861746936 ],
    CurrentAcceleration := [ 5180.079571404243, -9987.23908551058, 8369.828846550932 ],
    TargetPosition := [ 26.101611930284065, -62.69432172088365, -69.25146432081932 ],
    TargetVelocity := [ 0.0, 0.0, 0.0 ],
    TargetAcceleration := [ -131.90971166520217, -629.8496867961894, -805.129073987833 ]
  );
  
  positionExtrema : Struckig.PositionExtremaDesc;
END_VAR
TEST('Trajectory_HasMinDuration_HasTargetAcceleration_6');

ruckig();

// Check total duration of profiles
AssertEquals_LREAL(Expected := 10.0, Actual := ruckig.Duration, DELTA := 1E-8, Message := 'Duration incorrect');

// Check minimum duration
AssertEquals_LREAL(Expected := 10.0, Actual := ruckig.Duration, DELTA := 1E-8, Message := 'Duration incorrect');

// Check duration for each phase
positionExtrema := ruckig._profiles[0].positionExtrema();
AssertEquals_LREAL(0.0, positionExtrema.Tmax, 1E-9, message:='Profile[0] Tmax incorrect');
AssertEquals_LREAL(73.95774355738217, positionExtrema.Maximum, 1E-9, message:='Profile[0] maximum incorrect');
AssertEquals_LREAL(9.999670225720838, positionExtrema.Tmin, 1E-9, message:='Profile[0] Tmin incorrect');
AssertEquals_LREAL(26.101609539396815, positionExtrema.Minimum, 1E-9, message:='Profile[0] minimum incorrect');

positionExtrema := ruckig._profiles[1].positionExtrema();
AssertEquals_LREAL(0.0, positionExtrema.Tmax, 1E-9, message:='Profile[1] Tmax incorrect');
AssertEquals_LREAL(67.34262397589043, positionExtrema.Maximum, 1E-9, message:='Profile[1] maximum incorrect');
AssertEquals_LREAL(9.99842537578301, positionExtrema.Tmin, 1E-9, message:='Profile[1] Tmin incorrect');
AssertEquals_LREAL(-62.69458200011703, positionExtrema.Minimum, 1E-9, message:='Profile[1] minimum incorrect');

positionExtrema := ruckig._profiles[2].positionExtrema();
AssertEquals_LREAL(0.06090028897692612, positionExtrema.Tmax, 1E-9, message:='Profile[2] Tmax incorrect');
AssertEquals_LREAL(46.36974939931049, positionExtrema.Maximum, 1E-9, message:='Profile[2] maximum incorrect');
AssertEquals_LREAL(9.99798717731503, positionExtrema.Tmin, 1E-9, message:='Profile[2] Tmin incorrect');
AssertEquals_LREAL(-69.25200797820925, positionExtrema.Minimum, 1E-9, message:='Profile[2] minimum incorrect');
   

TEST_FINISHED();
END_METHOD

METHOD Test_Trajectory_HasMinDuration_HasTargetVelocity_16
VAR_INST
  ruckig : Struckig.Ruckig(0.001, 3) := (
  
    Synchronization := SynchronizationType.TimeSync,
    MinDuration := 7.0,
    MaxVelocity := [ 2000.0, 2000.0, 2000.0 ],
    MaxAcceleration := [ 20000.0, 20000.0, 20000.0 ],
    MaxJerk := [ 800000.0, 800000.0, 800000.0 ],
    CurrentPosition := [ 7.986268223464748, 30.66263768305589, -71.99998699577253 ],
    CurrentVelocity := [ -536.7319233815753, 166.5896044550318, 426.8037118862651 ],
    CurrentAcceleration := [ -3017.084283791076, -9424.883074091185, -1013.896197334474 ],
    TargetPosition := [ -34.478967783797216, 52.15227078186672, -24.73548276773934 ],
    TargetVelocity := [ -753.4402086481915, 518.6153002230694, -127.83329734668075 ],
    TargetAcceleration := [ 0.0, 0.0, 0.0 ]
  );
  
  positionExtrema : Struckig.PositionExtremaDesc;
END_VAR
TEST('Trajectory_HasMinDuration_HasTargetVelocity_16');

ruckig();

// Check total duration of profiles
AssertEquals_LREAL(Expected := 7.0, Actual := ruckig.Duration, DELTA := 1E-8, Message := 'Duration incorrect');

// Check minimum duration
AssertEquals_LREAL(Expected := 7.0, Actual := ruckig.Duration, DELTA := 1E-8, Message := 'Duration incorrect');

// Check duration for each phase
positionExtrema := ruckig._profiles[0].positionExtrema();
AssertEquals_LREAL(0.0, positionExtrema.Tmax, 1E-9, message:='Profile[0] Tmax incorrect');
AssertEquals_LREAL(7.986268223464748, positionExtrema.Maximum, 1E-9, message:='Profile[0] maximum incorrect');
AssertEquals_LREAL(7.000000000000001, positionExtrema.Tmin, 1E-9, message:='Profile[0] Tmin incorrect');
AssertEquals_LREAL(-34.478967783797216, positionExtrema.Minimum, 1E-9, message:='Profile[0] minimum incorrect');

positionExtrema := ruckig._profiles[1].positionExtrema();
AssertEquals_LREAL(7.000000000000002, positionExtrema.Tmax, 1E-9, message:='Profile[1] Tmax incorrect');
AssertEquals_LREAL(52.15227078186672, positionExtrema.Maximum, 1E-9, message:='Profile[1] maximum incorrect');
AssertEquals_LREAL(0.0, positionExtrema.Tmin, 1E-9, message:='Profile[1] Tmin incorrect');
AssertEquals_LREAL(30.66263768305589, positionExtrema.Minimum, 1E-9, message:='Profile[1] minimum incorrect');

positionExtrema := ruckig._profiles[2].positionExtrema();
AssertEquals_LREAL(6.97793366414829, positionExtrema.Tmax, 1E-9, message:='Profile[2] Tmax incorrect');
AssertEquals_LREAL(-23.14319435212213, positionExtrema.Maximum, 1E-9, message:='Profile[2] maximum incorrect');
AssertEquals_LREAL(0.0, positionExtrema.Tmin, 1E-9, message:='Profile[2] Tmin incorrect');
AssertEquals_LREAL(-71.99998699577253, positionExtrema.Minimum, 1E-9, message:='Profile[2] minimum incorrect');
   

TEST_FINISHED();
END_METHOD

METHOD Test_Trajectory_HasMinDuration_HasTargetVelocity_5
VAR_INST
  ruckig : Struckig.Ruckig(0.001, 3) := (
  
    Synchronization := SynchronizationType.TimeSync,
    MinDuration := 4.0,
    MaxVelocity := [ 2000.0, 2000.0, 2000.0 ],
    MaxAcceleration := [ 20000.0, 20000.0, 20000.0 ],
    MaxJerk := [ 800000.0, 800000.0, 800000.0 ],
    CurrentPosition := [ -3.497413438880301, 31.363081204112206, 63.367720727687384 ],
    CurrentVelocity := [ 866.434234141054, -171.78552231675485, 58.6036663712207 ],
    CurrentAcceleration := [ -6318.744631550888, -7187.849982760071, -3339.305374801589 ],
    TargetPosition := [ 53.47504800393719, 97.23185262639063, -88.75469905530662 ],
    TargetVelocity := [ 726.8020091222686, 210.07958633863836, 83.97764431780661 ],
    TargetAcceleration := [ 0.0, 0.0, 0.0 ]
  );
  
  positionExtrema : Struckig.PositionExtremaDesc;
END_VAR
TEST('Trajectory_HasMinDuration_HasTargetVelocity_5');

ruckig();

// Check total duration of profiles
AssertEquals_LREAL(Expected := 4.0, Actual := ruckig.Duration, DELTA := 1E-8, Message := 'Duration incorrect');

// Check minimum duration
AssertEquals_LREAL(Expected := 4.0, Actual := ruckig.Duration, DELTA := 1E-8, Message := 'Duration incorrect');

// Check duration for each phase
positionExtrema := ruckig._profiles[0].positionExtrema();
AssertEquals_LREAL(4.0, positionExtrema.Tmax, 1E-9, message:='Profile[0] Tmax incorrect');
AssertEquals_LREAL(53.47504800393719, positionExtrema.Maximum, 1E-9, message:='Profile[0] maximum incorrect');
AssertEquals_LREAL(0.0, positionExtrema.Tmin, 1E-9, message:='Profile[0] Tmin incorrect');
AssertEquals_LREAL(-3.497413438880301, positionExtrema.Minimum, 1E-9, message:='Profile[0] minimum incorrect');

positionExtrema := ruckig._profiles[1].positionExtrema();
AssertEquals_LREAL(3.9999999999999996, positionExtrema.Tmax, 1E-9, message:='Profile[1] Tmax incorrect');
AssertEquals_LREAL(97.23185262639063, positionExtrema.Maximum, 1E-9, message:='Profile[1] maximum incorrect');
AssertEquals_LREAL(0.03570009228167893, positionExtrema.Tmin, 1E-9, message:='Profile[1] Tmin incorrect');
AssertEquals_LREAL(26.442768005713322, positionExtrema.Minimum, 1E-9, message:='Profile[1] minimum incorrect');

positionExtrema := ruckig._profiles[2].positionExtrema();
AssertEquals_LREAL(0.00882488089698622, positionExtrema.Tmax, 1E-9, message:='Profile[2] Tmax incorrect');
AssertEquals_LREAL(63.66429252791513, positionExtrema.Maximum, 1E-9, message:='Profile[2] maximum incorrect');
AssertEquals_LREAL(3.98506688402464, positionExtrema.Tmin, 1E-9, message:='Profile[2] Tmin incorrect');
AssertEquals_LREAL(-89.5691863512788, positionExtrema.Minimum, 1E-9, message:='Profile[2] minimum incorrect');
   

TEST_FINISHED();
END_METHOD

METHOD Test_Trajectory_HasMinDuration_HasTargetVelocity_9
VAR_INST
  ruckig : Struckig.Ruckig(0.001, 3) := (
  
    Synchronization := SynchronizationType.TimeSync,
    MinDuration := 7.0,
    MaxVelocity := [ 2000.0, 2000.0, 2000.0 ],
    MaxAcceleration := [ 20000.0, 20000.0, 20000.0 ],
    MaxJerk := [ 800000.0, 800000.0, 800000.0 ],
    CurrentPosition := [ 32.77976315061471, 86.05945833221364, 34.11738301725197 ],
    CurrentVelocity := [ -981.2868512691955, 673.690792063916, -116.7982550185385 ],
    CurrentAcceleration := [ -4108.818774560344, 3339.252734800917, -7298.314365481016 ],
    TargetPosition := [ -55.314233526195245, 80.34443440826854, -61.91751423362351 ],
    TargetVelocity := [ 817.0398878216338, -103.40219473844786, -439.1476692838428 ],
    TargetAcceleration := [ 0.0, 0.0, 0.0 ]
  );
  
  positionExtrema : Struckig.PositionExtremaDesc;
END_VAR
TEST('Trajectory_HasMinDuration_HasTargetVelocity_9');

ruckig();

// Check total duration of profiles
AssertEquals_LREAL(Expected := 7.0, Actual := ruckig.Duration, DELTA := 1E-8, Message := 'Duration incorrect');

// Check minimum duration
AssertEquals_LREAL(Expected := 7.0, Actual := ruckig.Duration, DELTA := 1E-8, Message := 'Duration incorrect');

// Check duration for each phase
positionExtrema := ruckig._profiles[0].positionExtrema();
AssertEquals_LREAL(0.0, positionExtrema.Tmax, 1E-9, message:='Profile[0] Tmax incorrect');
AssertEquals_LREAL(32.77976315061471, positionExtrema.Maximum, 1E-9, message:='Profile[0] maximum incorrect');
AssertEquals_LREAL(6.938765999899139, positionExtrema.Tmin, 1E-9, message:='Profile[0] Tmin incorrect');
AssertEquals_LREAL(-82.11714814813035, positionExtrema.Minimum, 1E-9, message:='Profile[0] minimum incorrect');

positionExtrema := ruckig._profiles[1].positionExtrema();
AssertEquals_LREAL(0.060258152451987596, positionExtrema.Tmax, 1E-9, message:='Profile[1] Tmax incorrect');
AssertEquals_LREAL(108.93997970698679, positionExtrema.Maximum, 1E-9, message:='Profile[1] maximum incorrect');
AssertEquals_LREAL(7.0, positionExtrema.Tmin, 1E-9, message:='Profile[1] Tmin incorrect');
AssertEquals_LREAL(80.34443440826854, positionExtrema.Minimum, 1E-9, message:='Profile[1] minimum incorrect');

positionExtrema := ruckig._profiles[2].positionExtrema();
AssertEquals_LREAL(0.0, positionExtrema.Tmax, 1E-9, message:='Profile[2] Tmax incorrect');
AssertEquals_LREAL(34.11738301725197, positionExtrema.Maximum, 1E-9, message:='Profile[2] maximum incorrect');
AssertEquals_LREAL(7.0, positionExtrema.Tmin, 1E-9, message:='Profile[2] Tmin incorrect');
AssertEquals_LREAL(-61.91751423362351, positionExtrema.Minimum, 1E-9, message:='Profile[2] minimum incorrect');
   

TEST_FINISHED();
END_METHOD

METHOD Test_Trajectory_HasMinDuration_HasTargetVelocity_HasTargetAcceleration_10
VAR_INST
  ruckig : Struckig.Ruckig(0.001, 3) := (
  
    Synchronization := SynchronizationType.TimeSync,
    MinDuration := 5.0,
    MaxVelocity := [ 2000.0, 2000.0, 2000.0 ],
    MaxAcceleration := [ 20000.0, 20000.0, 20000.0 ],
    MaxJerk := [ 800000.0, 800000.0, 800000.0 ],
    CurrentPosition := [ -63.70257714146867, 22.730031520740937, -51.56243568859453 ],
    CurrentVelocity := [ -520.8565160201103, 365.56449403589454, 835.823452928573 ],
    CurrentAcceleration := [ 9598.328373658613, -2893.4545241775922, 121.46690068480166 ],
    TargetPosition := [ 22.750797061424464, 74.13128623236747, 69.96760822932885 ],
    TargetVelocity := [ -174.7936793360849, -636.488954459087, -938.8757724326924 ],
    TargetAcceleration := [ 391.8907382899415, -699.6872603922127, 978.1856283310506 ]
  );
  
  positionExtrema : Struckig.PositionExtremaDesc;
END_VAR
TEST('Trajectory_HasMinDuration_HasTargetVelocity_HasTargetAcceleration_10');

ruckig();

// Check total duration of profiles
AssertEquals_LREAL(Expected := 5.0, Actual := ruckig.Duration, DELTA := 1E-8, Message := 'Duration incorrect');

// Check minimum duration
AssertEquals_LREAL(Expected := 5.0, Actual := ruckig.Duration, DELTA := 1E-8, Message := 'Duration incorrect');

// Check duration for each phase
positionExtrema := ruckig._profiles[0].positionExtrema();
AssertEquals_LREAL(4.975346883096284, positionExtrema.Tmax, 1E-9, message:='Profile[0] Tmax incorrect');
AssertEquals_LREAL(25.348702524320338, positionExtrema.Maximum, 1E-9, message:='Profile[0] maximum incorrect');
AssertEquals_LREAL(0.0358766442937755, positionExtrema.Tmin, 1E-9, message:='Profile[0] Tmin incorrect');
AssertEquals_LREAL(-72.4234881857976, positionExtrema.Minimum, 1E-9, message:='Profile[0] minimum incorrect');

positionExtrema := ruckig._profiles[1].positionExtrema();
AssertEquals_LREAL(4.949024471203024, positionExtrema.Tmax, 1E-9, message:='Profile[1] Tmax incorrect');
AssertEquals_LREAL(91.55742573849955, positionExtrema.Maximum, 1E-9, message:='Profile[1] maximum incorrect');
AssertEquals_LREAL(0.0, positionExtrema.Tmin, 1E-9, message:='Profile[1] Tmin incorrect');
AssertEquals_LREAL(22.730031520740937, positionExtrema.Minimum, 1E-9, message:='Profile[1] minimum incorrect');

positionExtrema := ruckig._profiles[2].positionExtrema();
AssertEquals_LREAL(4.933596685985829, positionExtrema.Tmax, 1E-9, message:='Profile[2] Tmax incorrect');
AssertEquals_LREAL(104.72094552143355, positionExtrema.Maximum, 1E-9, message:='Profile[2] maximum incorrect');
AssertEquals_LREAL(0.0, positionExtrema.Tmin, 1E-9, message:='Profile[2] Tmin incorrect');
AssertEquals_LREAL(-51.56243568859453, positionExtrema.Minimum, 1E-9, message:='Profile[2] minimum incorrect');
   

TEST_FINISHED();
END_METHOD

METHOD Test_Trajectory_HasMinDuration_HasTargetVelocity_HasTargetAcceleration_12
VAR_INST
  ruckig : Struckig.Ruckig(0.001, 3) := (
  
    Synchronization := SynchronizationType.TimeSync,
    MinDuration := 8.0,
    MaxVelocity := [ 2000.0, 2000.0, 2000.0 ],
    MaxAcceleration := [ 20000.0, 20000.0, 20000.0 ],
    MaxJerk := [ 800000.0, 800000.0, 800000.0 ],
    CurrentPosition := [ 34.32407664987838, -19.61426768221135, 0.08400152186804632 ],
    CurrentVelocity := [ -637.0909066222588, -315.93942928026286, -768.0946853095916 ],
    CurrentAcceleration := [ 5239.657334131169, -3857.903449466051, 5261.930344314516 ],
    TargetPosition := [ -0.6332298839860186, 7.05929814872006, 84.95032201129774 ],
    TargetVelocity := [ -688.3030057720259, 935.2283186121415, -773.3660434214753 ],
    TargetAcceleration := [ 75.12349151093213, -861.2904239623496, 251.41067093552897 ]
  );
  
  positionExtrema : Struckig.PositionExtremaDesc;
END_VAR
TEST('Trajectory_HasMinDuration_HasTargetVelocity_HasTargetAcceleration_12');

ruckig();

// Check total duration of profiles
AssertEquals_LREAL(Expected := 8.0, Actual := ruckig.Duration, DELTA := 1E-8, Message := 'Duration incorrect');

// Check minimum duration
AssertEquals_LREAL(Expected := 8.0, Actual := ruckig.Duration, DELTA := 1E-8, Message := 'Duration incorrect');

// Check duration for each phase
positionExtrema := ruckig._profiles[0].positionExtrema();
AssertEquals_LREAL(0.0, positionExtrema.Tmax, 1E-9, message:='Profile[0] Tmax incorrect');
AssertEquals_LREAL(34.32407664987838, positionExtrema.Maximum, 1E-9, message:='Profile[0] maximum incorrect');
AssertEquals_LREAL(8.0, positionExtrema.Tmin, 1E-9, message:='Profile[0] Tmin incorrect');
AssertEquals_LREAL(-0.6332298839860186, positionExtrema.Minimum, 1E-9, message:='Profile[0] minimum incorrect');

positionExtrema := ruckig._profiles[1].positionExtrema();
AssertEquals_LREAL(8.0, positionExtrema.Tmax, 1E-9, message:='Profile[1] Tmax incorrect');
AssertEquals_LREAL(7.05929814872006, positionExtrema.Maximum, 1E-9, message:='Profile[1] maximum incorrect');
AssertEquals_LREAL(0.04490272145795441, positionExtrema.Tmin, 1E-9, message:='Profile[1] Tmin incorrect');
AssertEquals_LREAL(-27.725399337897105, positionExtrema.Minimum, 1E-9, message:='Profile[1] minimum incorrect');

positionExtrema := ruckig._profiles[2].positionExtrema();
AssertEquals_LREAL(7.941603003365496, positionExtrema.Tmax, 1E-9, message:='Profile[2] Tmax incorrect');
AssertEquals_LREAL(109.67291667846435, positionExtrema.Maximum, 1E-9, message:='Profile[2] maximum incorrect');
AssertEquals_LREAL(0.05210502444806486, positionExtrema.Tmin, 1E-9, message:='Profile[2] Tmin incorrect');
AssertEquals_LREAL(-19.88492411775111, positionExtrema.Minimum, 1E-9, message:='Profile[2] minimum incorrect');
   

TEST_FINISHED();
END_METHOD

METHOD Test_Trajectory_HasMinDuration_HasTargetVelocity_HasTargetAcceleration_15
VAR_INST
  ruckig : Struckig.Ruckig(0.001, 3) := (
  
    Synchronization := SynchronizationType.TimeSync,
    MinDuration := 6.0,
    MaxVelocity := [ 2000.0, 2000.0, 2000.0 ],
    MaxAcceleration := [ 20000.0, 20000.0, 20000.0 ],
    MaxJerk := [ 800000.0, 800000.0, 800000.0 ],
    CurrentPosition := [ 80.29599725108966, -16.595240167642288, -10.563218674718456 ],
    CurrentVelocity := [ -665.2939916748119, -252.31162160327165, 910.7605496896838 ],
    CurrentAcceleration := [ -6038.086221066726, 5702.712022046548, -5391.38537360544 ],
    TargetPosition := [ -15.947396233027035, -52.93402548041466, -99.24861248238838 ],
    TargetVelocity := [ -82.3068299752083, 810.5242632500622, -475.5452525569576 ],
    TargetAcceleration := [ 797.6779209006231, 304.9451091028675, 294.8876599912337 ]
  );
  
  positionExtrema : Struckig.PositionExtremaDesc;
END_VAR
TEST('Trajectory_HasMinDuration_HasTargetVelocity_HasTargetAcceleration_15');

ruckig();

// Check total duration of profiles
AssertEquals_LREAL(Expected := 6.0, Actual := ruckig.Duration, DELTA := 1E-8, Message := 'Duration incorrect');

// Check minimum duration
AssertEquals_LREAL(Expected := 6.0, Actual := ruckig.Duration, DELTA := 1E-8, Message := 'Duration incorrect');

// Check duration for each phase
positionExtrema := ruckig._profiles[0].positionExtrema();
AssertEquals_LREAL(0.0, positionExtrema.Tmax, 1E-9, message:='Profile[0] Tmax incorrect');
AssertEquals_LREAL(80.29599725108966, positionExtrema.Maximum, 1E-9, message:='Profile[0] maximum incorrect');
AssertEquals_LREAL(5.999999999999999, positionExtrema.Tmin, 1E-9, message:='Profile[0] Tmin incorrect');
AssertEquals_LREAL(-15.947396233027035, positionExtrema.Minimum, 1E-9, message:='Profile[0] minimum incorrect');

positionExtrema := ruckig._profiles[1].positionExtrema();
AssertEquals_LREAL(0.0, positionExtrema.Tmax, 1E-9, message:='Profile[1] Tmax incorrect');
AssertEquals_LREAL(-16.595240167642288, positionExtrema.Maximum, 1E-9, message:='Profile[1] maximum incorrect');
AssertEquals_LREAL(5.939358209422553, positionExtrema.Tmin, 1E-9, message:='Profile[1] Tmin incorrect');
AssertEquals_LREAL(-79.08901602854112, positionExtrema.Minimum, 1E-9, message:='Profile[1] minimum incorrect');

positionExtrema := ruckig._profiles[2].positionExtrema();
AssertEquals_LREAL(0.058957419609001596, positionExtrema.Tmax, 1E-9, message:='Profile[2] Tmax incorrect');
AssertEquals_LREAL(16.2518405159937, positionExtrema.Maximum, 1E-9, message:='Profile[2] maximum incorrect');
AssertEquals_LREAL(6.0, positionExtrema.Tmin, 1E-9, message:='Profile[2] Tmin incorrect');
AssertEquals_LREAL(-99.24861248238838, positionExtrema.Minimum, 1E-9, message:='Profile[2] minimum incorrect');
   

TEST_FINISHED();
END_METHOD

METHOD Test_Trajectory_HasMinDuration_HasTargetVelocity_HasTargetAcceleration_18
VAR_INST
  ruckig : Struckig.Ruckig(0.001, 3) := (
  
    Synchronization := SynchronizationType.TimeSync,
    MinDuration := 6.0,
    MaxVelocity := [ 2000.0, 2000.0, 2000.0 ],
    MaxAcceleration := [ 20000.0, 20000.0, 20000.0 ],
    MaxJerk := [ 800000.0, 800000.0, 800000.0 ],
    CurrentPosition := [ 81.8189456654396, -34.648960679925025, -51.77657021421829 ],
    CurrentVelocity := [ 52.71918271967047, -512.6427429671598, 347.52161587573437 ],
    CurrentAcceleration := [ -463.2079718295354, -9185.891702573537, 7766.274147421525 ],
    TargetPosition := [ 28.57172398615708, 23.600629576782865, -2.4216248210818776 ],
    TargetVelocity := [ 159.80128500214232, -165.6494233580952, 407.13274543851867 ],
    TargetAcceleration := [ -496.57312685360756, 646.2561464861296, 884.0412488799539 ]
  );
  
  positionExtrema : Struckig.PositionExtremaDesc;
END_VAR
TEST('Trajectory_HasMinDuration_HasTargetVelocity_HasTargetAcceleration_18');

ruckig();

// Check total duration of profiles
AssertEquals_LREAL(Expected := 6.0, Actual := ruckig.Duration, DELTA := 1E-8, Message := 'Duration incorrect');

// Check minimum duration
AssertEquals_LREAL(Expected := 6.0, Actual := ruckig.Duration, DELTA := 1E-8, Message := 'Duration incorrect');

// Check duration for each phase
positionExtrema := ruckig._profiles[0].positionExtrema();
AssertEquals_LREAL(0.012217427498857257, positionExtrema.Tmax, 1E-9, message:='Profile[0] Tmax incorrect');
AssertEquals_LREAL(82.2020759262068, positionExtrema.Maximum, 1E-9, message:='Profile[0] maximum incorrect');
AssertEquals_LREAL(5.975125497966807, positionExtrema.Tmin, 1E-9, message:='Profile[0] Tmin incorrect');
AssertEquals_LREAL(26.251513510769477, positionExtrema.Minimum, 1E-9, message:='Profile[0] minimum incorrect');

positionExtrema := ruckig._profiles[1].positionExtrema();
AssertEquals_LREAL(5.9750978983936935, positionExtrema.Tmax, 1E-9, message:='Profile[1] Tmax incorrect');
AssertEquals_LREAL(26.068274316521368, positionExtrema.Maximum, 1E-9, message:='Profile[1] maximum incorrect');
AssertEquals_LREAL(0.059557771163129256, positionExtrema.Tmin, 1E-9, message:='Profile[1] Tmin incorrect');
AssertEquals_LREAL(-55.87398334808502, positionExtrema.Minimum, 1E-9, message:='Profile[1] minimum incorrect');

positionExtrema := ruckig._profiles[2].positionExtrema();
AssertEquals_LREAL(6.0, positionExtrema.Tmax, 1E-9, message:='Profile[2] Tmax incorrect');
AssertEquals_LREAL(-2.4216248210818776, positionExtrema.Maximum, 1E-9, message:='Profile[2] maximum incorrect');
AssertEquals_LREAL(0.0, positionExtrema.Tmin, 1E-9, message:='Profile[2] Tmin incorrect');
AssertEquals_LREAL(-51.77657021421829, positionExtrema.Minimum, 1E-9, message:='Profile[2] minimum incorrect');
   

TEST_FINISHED();
END_METHOD

METHOD Test_Trajectory_HasMinDuration_HasTargetVelocity_HasTargetAcceleration_20
VAR_INST
  ruckig : Struckig.Ruckig(0.001, 3) := (
  
    Synchronization := SynchronizationType.TimeSync,
    MinDuration := 1.0,
    MaxVelocity := [ 2000.0, 2000.0, 2000.0 ],
    MaxAcceleration := [ 20000.0, 20000.0, 20000.0 ],
    MaxJerk := [ 800000.0, 800000.0, 800000.0 ],
    CurrentPosition := [ 74.13037097871606, 50.87684992213954, -35.461969837009065 ],
    CurrentVelocity := [ -104.6717721730954, 978.8741284865525, 932.4293320305519 ],
    CurrentAcceleration := [ -1484.1311843071398, -3303.1671799903806, -254.44992328560875 ],
    TargetPosition := [ -53.87981386222778, -79.63304774882201, 29.944494194232874 ],
    TargetVelocity := [ -444.5052876664206, 76.57672906373682, 439.3701152281369 ],
    TargetAcceleration := [ 223.1822145745084, 144.20762241820466, 871.7177536324762 ]
  );
  
  positionExtrema : Struckig.PositionExtremaDesc;
END_VAR
TEST('Trajectory_HasMinDuration_HasTargetVelocity_HasTargetAcceleration_20');

ruckig();

// Check total duration of profiles
AssertEquals_LREAL(Expected := 1.0, Actual := ruckig.Duration, DELTA := 1E-8, Message := 'Duration incorrect');

// Check minimum duration
AssertEquals_LREAL(Expected := 1.0, Actual := ruckig.Duration, DELTA := 1E-8, Message := 'Duration incorrect');

// Check duration for each phase
positionExtrema := ruckig._profiles[0].positionExtrema();
AssertEquals_LREAL(0.0, positionExtrema.Tmax, 1E-9, message:='Profile[0] Tmax incorrect');
AssertEquals_LREAL(74.13037097871606, positionExtrema.Maximum, 1E-9, message:='Profile[0] maximum incorrect');
AssertEquals_LREAL(1.0, positionExtrema.Tmin, 1E-9, message:='Profile[0] Tmin incorrect');
AssertEquals_LREAL(-53.87981386222778, positionExtrema.Minimum, 1E-9, message:='Profile[0] minimum incorrect');

positionExtrema := ruckig._profiles[1].positionExtrema();
AssertEquals_LREAL(0.05795449228928962, positionExtrema.Tmax, 1E-9, message:='Profile[1] Tmax incorrect');
AssertEquals_LREAL(82.91327789055885, positionExtrema.Maximum, 1E-9, message:='Profile[1] maximum incorrect');
AssertEquals_LREAL(0.9863428350510189, positionExtrema.Tmin, 1E-9, message:='Profile[1] Tmin incorrect');
AssertEquals_LREAL(-80.32577887227478, positionExtrema.Minimum, 1E-9, message:='Profile[1] minimum incorrect');

positionExtrema := ruckig._profiles[2].positionExtrema();
AssertEquals_LREAL(1.0, positionExtrema.Tmax, 1E-9, message:='Profile[2] Tmax incorrect');
AssertEquals_LREAL(29.944494194232874, positionExtrema.Maximum, 1E-9, message:='Profile[2] maximum incorrect');
AssertEquals_LREAL(0.0, positionExtrema.Tmin, 1E-9, message:='Profile[2] Tmin incorrect');
AssertEquals_LREAL(-35.461969837009065, positionExtrema.Minimum, 1E-9, message:='Profile[2] minimum incorrect');
   

TEST_FINISHED();
END_METHOD

END_FUNCTION_BLOCK

// ---- POUs/TargetPosTest.TcPOU
FUNCTION_BLOCK TargetPosTest EXTENDS TcUnit.FB_TestSuite
VAR
  ruckig : Struckig.Ruckig(0.001, 3) := (
  
    Synchronization := SynchronizationType.TimeSync,        
    MaxVelocity := [ 2000.00000000000000000000, 2000.00000000000000000000, 2000.00000000000000000000 ],
    MaxAcceleration := [ 20000.00000000000000000000, 20000.00000000000000000000, 20000.00000000000000000000 ],
    MaxJerk := [ 800000.00000000000000000000, 800000.00000000000000000000, 800000.00000000000000000000 ],
    CurrentPosition := [ 48.86656216713086564596, 31.55963588984187140341, -13.09422790776093847853 ],
    CurrentVelocity := [ -274.21841080128081102885, -440.94461360926254656079, -764.75678162210920163488 ],
    CurrentAcceleration := [ -1478.09700836416959646158, 686.79611869591644790489, -9263.72976579731221136171 ],
    TargetPosition := [ 25.57994474955607699940, -15.83091418217283319336, -38.97164514571973370494 ],
    TargetVelocity := [ 0.00000000000000000000, 0.00000000000000000000, 0.00000000000000000000 ],
    TargetAcceleration := [ 0.00000000000000000000, 0.00000000000000000000, 0.00000000000000000000 ]
  );
  
  positionExtrema : Struckig.PositionExtremaDesc;  
END_VAR

Test_Trajectory_2();;
Test_Trajectory_5();
Test_Trajectory_6();
Test_Trajectory_7();
Test_Trajectory_12();
Test_Trajectory_16(); // this test required to do a more precise implementation of cbrt
Test_Trajectory_30();
Test_Trajectory_32();
Test_Trajectory_33();
Test_Trajectory_40();
Test_Trajectory_49();
Test_Trajectory_53();
Test_Trajectory_59();
Test_Trajectory_62();
Test_Trajectory_64();
Test_Trajectory_65();
Test_Trajectory_68();

METHOD Test_Trajectory_12
VAR_INST
  ruckig : Struckig.Ruckig(0.001, 3) := (
  
    Synchronization := SynchronizationType.TimeSync,        
    MaxVelocity := [ 2000.00000000000000000000, 2000.00000000000000000000, 2000.00000000000000000000 ],
    MaxAcceleration := [ 20000.00000000000000000000, 20000.00000000000000000000, 20000.00000000000000000000 ],
    MaxJerk := [ 800000.00000000000000000000, 800000.00000000000000000000, 800000.00000000000000000000 ],
    CurrentPosition := [ 12.15863849634686744139, 83.56438022017914590833, -29.82534868849941744884 ],
    CurrentVelocity := [ -881.54677264260010360886, -40.22247547933807254594, 795.30816871835008896596 ],
    CurrentAcceleration := [ 6802.73049394882036722265, -2844.95338607063877134351, -3652.21806306270900677191 ],
    TargetPosition := [ 61.24855302996508044089, -54.65891429617437324850, 65.64407005892678625969 ],
    TargetVelocity := [ 0.00000000000000000000, 0.00000000000000000000, 0.00000000000000000000 ],
    TargetAcceleration := [ 0.00000000000000000000, 0.00000000000000000000, 0.00000000000000000000 ]
  );
  
  positionExtrema : Struckig.PositionExtremaDesc;
END_VAR
TEST('Trajectory_12');

ruckig();

// Check total duration of profiles
AssertEquals_LREAL(Expected := 0.18765626933931714437, Actual := ruckig.Duration, DELTA := 1E-8, Message := 'Duration incorrect');

// Check duration for each phase
positionExtrema := ruckig._profiles[0].positionExtrema();
AssertEquals_LREAL(0.18765626933931711662, positionExtrema.Tmax, 1E-9, message:='Profile[0] Tmax incorrect');
AssertEquals_LREAL(61.24855302996508044089, positionExtrema.Maximum, 1E-9, message:='Profile[0] maximum incorrect');
AssertEquals_LREAL(0.01649658688256397387, positionExtrema.Tmin, 1E-9, message:='Profile[0] Tmin incorrect');
AssertEquals_LREAL(-0.85965741863935996037, positionExtrema.Minimum, 1E-9, message:='Profile[0] minimum incorrect');

positionExtrema := ruckig._profiles[1].positionExtrema();
AssertEquals_LREAL(0.00000000000000000000, positionExtrema.Tmax, 1E-9, message:='Profile[1] Tmax incorrect');
AssertEquals_LREAL(83.56438022017914590833, positionExtrema.Maximum, 1E-9, message:='Profile[1] maximum incorrect');
AssertEquals_LREAL(0.18765626933931714437, positionExtrema.Tmin, 1E-9, message:='Profile[1] Tmin incorrect');
AssertEquals_LREAL(-54.65891429617437324850, positionExtrema.Minimum, 1E-9, message:='Profile[1] minimum incorrect');

positionExtrema := ruckig._profiles[2].positionExtrema();
AssertEquals_LREAL(0.18765626933931711662, positionExtrema.Tmax, 1E-9, message:='Profile[2] Tmax incorrect');
AssertEquals_LREAL(65.64407005892678625969, positionExtrema.Maximum, 1E-9, message:='Profile[2] maximum incorrect');
AssertEquals_LREAL(0.00000000000000000000, positionExtrema.Tmin, 1E-9, message:='Profile[2] Tmin incorrect');
AssertEquals_LREAL(-29.82534868849941744884, positionExtrema.Minimum, 1E-9, message:='Profile[2] minimum incorrect');
   

TEST_FINISHED();
END_METHOD

METHOD Test_Trajectory_16
VAR_INST
  ruckig : Struckig.Ruckig(0.001, 3) := (
  
    Synchronization := SynchronizationType.TimeSync,        
    MaxVelocity := [ 2000.00000000000000000000, 2000.00000000000000000000, 2000.00000000000000000000 ],
    MaxAcceleration := [ 20000.00000000000000000000, 20000.00000000000000000000, 20000.00000000000000000000 ],
    MaxJerk := [ 800000.00000000000000000000, 800000.00000000000000000000, 800000.00000000000000000000 ],
    CurrentPosition := [ 8.21667911707363884943, -42.91905125747626215116, 48.44417367414695263506 ],
    CurrentVelocity := [ -786.82135287550590874162, 724.24582523622666485608, -678.96507198447488917736 ],
    CurrentAcceleration := [ 2775.55640569175011478364, 5006.65330127050037845038, -1991.17849814757664717035 ],
    TargetPosition := [ -91.18523630560480341956, 39.65724384459844031880, 80.00859285567460688071 ],
    TargetVelocity := [ 0.00000000000000000000, 0.00000000000000000000, 0.00000000000000000000 ],
    TargetAcceleration := [ 0.00000000000000000000, 0.00000000000000000000, 0.00000000000000000000 ]
  );
  
  positionExtrema : Struckig.PositionExtremaDesc;
END_VAR
TEST('Trajectory_16');

ruckig();

// Check total duration of profiles
AssertEquals_LREAL(Expected := 0.16787256653000462436, Actual := ruckig.Duration, DELTA := 1E-8, Message := 'Duration incorrect');

// Check duration for each phase
positionExtrema := ruckig._profiles[0].positionExtrema();
AssertEquals_LREAL(0, positionExtrema.Tmax, 1E-9, message:='Profile[0] Tmax incorrect');
AssertEquals_LREAL(8.2166791170736388494, positionExtrema.Maximum, 1E-9, message:='Profile[0] maximum incorrect');
AssertEquals_LREAL(0.16787256653000462436, positionExtrema.Tmin, 1E-9, message:='Profile[0] Tmin incorrect');
AssertEquals_LREAL(-91.18523630560480342, positionExtrema.Minimum, 1E-9, message:='Profile[0] minimum incorrect');

positionExtrema := ruckig._profiles[1].positionExtrema();
AssertEquals_LREAL(0.16787256609842091115, positionExtrema.Tmax, 1E-9, message:='Profile[1] Tmax incorrect');
AssertEquals_LREAL(39.657243844598482951, positionExtrema.Maximum, 1E-9, message:='Profile[1] maximum incorrect');
AssertEquals_LREAL(0, positionExtrema.Tmin, 1E-9, message:='Profile[1] Tmin incorrect');
AssertEquals_LREAL(-42.919051257476262151, positionExtrema.Minimum, 1E-9, message:='Profile[1] minimum incorrect');

positionExtrema := ruckig._profiles[2].positionExtrema();
AssertEquals_LREAL(0.16787256609842091115, positionExtrema.Tmax, 1E-9, message:='Profile[2] Tmax incorrect');
AssertEquals_LREAL(80.008592855674606881, positionExtrema.Maximum, 1E-9, message:='Profile[2] maximum incorrect');
AssertEquals_LREAL(0.027488973122684470102, positionExtrema.Tmin, 1E-9, message:='Profile[2] Tmin incorrect');
AssertEquals_LREAL(31.797392745296477301, positionExtrema.Minimum, 1E-9, message:='Profile[2] minimum incorrect');
   

TEST_FINISHED();
END_METHOD

METHOD Test_Trajectory_2
VAR_INST
  ruckig : Struckig.Ruckig(0.001, 3) := (
  
    Synchronization := SynchronizationType.TimeSync,        
    MaxVelocity := [ 2000.00000000000000000000, 2000.00000000000000000000, 2000.00000000000000000000 ],
    MaxAcceleration := [ 20000.00000000000000000000, 20000.00000000000000000000, 20000.00000000000000000000 ],
    MaxJerk := [ 800000.00000000000000000000, 800000.00000000000000000000, 800000.00000000000000000000 ],
    CurrentPosition := [ 44.74559775494429914033, 63.66880079927278757168, -12.48356919175202506267 ],
    CurrentVelocity := [ 264.84303106023071450181, -712.27423462239960372244, -643.21373646696986270399 ],
    CurrentAcceleration := [ 424.20358939641846518498, -6495.14198884339384676423, -9831.31287541736855928320 ],
    TargetPosition := [ 57.39429753248339238780, 42.08707495871314563374, -1.97763153852878303951 ],
    TargetVelocity := [ 0.00000000000000000000, 0.00000000000000000000, 0.00000000000000000000 ],
    TargetAcceleration := [ 0.00000000000000000000, 0.00000000000000000000, 0.00000000000000000000 ]
  );
  
  positionExtrema : Struckig.PositionExtremaDesc;
END_VAR
TEST('Trajectory_2');

ruckig();

// Check total duration of profiles
AssertEquals_LREAL(Expected := 0.16542491911229942336, Actual := ruckig.Duration, DELTA := 1E-8, Message := 'Duration incorrect');

// Check duration for each phase
positionExtrema := ruckig._profiles[0].positionExtrema();
AssertEquals_LREAL(0.16542491892541816290, positionExtrema.Tmax, 1E-9, message:='Profile[0] Tmax incorrect');
AssertEquals_LREAL(57.39429753248339949323, positionExtrema.Maximum, 1E-9, message:='Profile[0] maximum incorrect');
AssertEquals_LREAL(0.00000000000000000000, positionExtrema.Tmin, 1E-9, message:='Profile[0] Tmin incorrect');
AssertEquals_LREAL(44.74559775494429914033, positionExtrema.Minimum, 1E-9, message:='Profile[0] minimum incorrect');

positionExtrema := ruckig._profiles[1].positionExtrema();
AssertEquals_LREAL(0.00000000000000000000, positionExtrema.Tmax, 1E-9, message:='Profile[1] Tmax incorrect');
AssertEquals_LREAL(63.66880079927278757168, positionExtrema.Maximum, 1E-9, message:='Profile[1] maximum incorrect');
AssertEquals_LREAL(0.06011117382266835396, positionExtrema.Tmin, 1E-9, message:='Profile[1] Tmin incorrect');
AssertEquals_LREAL(35.26367745920458673936, positionExtrema.Minimum, 1E-9, message:='Profile[1] minimum incorrect');

positionExtrema := ruckig._profiles[2].positionExtrema();
AssertEquals_LREAL(0.16542491911229942336, positionExtrema.Tmax, 1E-9, message:='Profile[2] Tmax incorrect');
AssertEquals_LREAL(-1.97763153852878303951, positionExtrema.Maximum, 1E-9, message:='Profile[2] maximum incorrect');
AssertEquals_LREAL(0.08144760340330899073, positionExtrema.Tmin, 1E-9, message:='Profile[2] Tmin incorrect');
AssertEquals_LREAL(-36.92186481482234938767, positionExtrema.Minimum, 1E-9, message:='Profile[2] minimum incorrect');
   

TEST_FINISHED();
END_METHOD

METHOD Test_Trajectory_30
VAR_INST
  ruckig : Struckig.Ruckig(0.001, 3) := (
  
    Synchronization := SynchronizationType.TimeSync,        
    MaxVelocity := [ 2000.00000000000000000000, 2000.00000000000000000000, 2000.00000000000000000000 ],
    MaxAcceleration := [ 20000.00000000000000000000, 20000.00000000000000000000, 20000.00000000000000000000 ],
    MaxJerk := [ 800000.00000000000000000000, 800000.00000000000000000000, 800000.00000000000000000000 ],
    CurrentPosition := [ 20.18249544120934046987, -10.33662927823941402039, -59.33613032688207766796 ],
    CurrentVelocity := [ -147.36941969263784812938, 276.37127321170169125253, -471.16528659637026521523 ],
    CurrentAcceleration := [ 5958.91709773212642176077, -6024.30381588076943444321, 4027.41742253926349803805 ],
    TargetPosition := [ 57.35278694063060811459, 37.88908861774962133495, 47.84009680376084361342 ],
    TargetVelocity := [ 0.00000000000000000000, 0.00000000000000000000, 0.00000000000000000000 ],
    TargetAcceleration := [ 0.00000000000000000000, 0.00000000000000000000, 0.00000000000000000000 ]
  );
  
  positionExtrema : Struckig.PositionExtremaDesc;
END_VAR
TEST('Trajectory_30');

ruckig();

// Check total duration of profiles
AssertEquals_LREAL(Expected := 0.19875826019833076064, Actual := ruckig.Duration, DELTA := 1E-8, Message := 'Duration incorrect');

// Check duration for each phase
positionExtrema := ruckig._profiles[0].positionExtrema();
AssertEquals_LREAL(0.19875826019833078839, positionExtrema.Tmax, 1E-9, message:='Profile[0] Tmax incorrect');
AssertEquals_LREAL(57.35278694063060811459, positionExtrema.Maximum, 1E-9, message:='Profile[0] maximum incorrect');
AssertEquals_LREAL(0.01314032839612196309, positionExtrema.Tmin, 1E-9, message:='Profile[0] Tmin incorrect');
AssertEquals_LREAL(19.06299300602372071012, positionExtrema.Minimum, 1E-9, message:='Profile[0] minimum incorrect');

positionExtrema := ruckig._profiles[1].positionExtrema();
AssertEquals_LREAL(0.19875826019833076064, positionExtrema.Tmax, 1E-9, message:='Profile[1] Tmax incorrect');
AssertEquals_LREAL(37.88908861774962133495, positionExtrema.Maximum, 1E-9, message:='Profile[1] maximum incorrect');
AssertEquals_LREAL(0.00000000000000000000, positionExtrema.Tmin, 1E-9, message:='Profile[1] Tmin incorrect');
AssertEquals_LREAL(-10.33662927823941402039, positionExtrema.Minimum, 1E-9, message:='Profile[1] minimum incorrect');

positionExtrema := ruckig._profiles[2].positionExtrema();
AssertEquals_LREAL(0.19875826019833076064, positionExtrema.Tmax, 1E-9, message:='Profile[2] Tmax incorrect');
AssertEquals_LREAL(47.84009680376084361342, positionExtrema.Maximum, 1E-9, message:='Profile[2] maximum incorrect');
AssertEquals_LREAL(0.01996572822182592077, positionExtrema.Tmin, 1E-9, message:='Profile[2] Tmin incorrect');
AssertEquals_LREAL(-66.87937049880544293501, positionExtrema.Minimum, 1E-9, message:='Profile[2] minimum incorrect');
   

TEST_FINISHED();
END_METHOD

METHOD Test_Trajectory_32
VAR_INST
  ruckig : Struckig.Ruckig(0.001, 3) := (
  
    Synchronization := SynchronizationType.TimeSync,        
    MaxVelocity := [ 2000.00000000000000000000, 2000.00000000000000000000, 2000.00000000000000000000 ],
    MaxAcceleration := [ 20000.00000000000000000000, 20000.00000000000000000000, 20000.00000000000000000000 ],
    MaxJerk := [ 800000.00000000000000000000, 800000.00000000000000000000, 800000.00000000000000000000 ],
    CurrentPosition := [ -71.32072487430589546875, 75.77874394332496876814, -31.17619673281745917848 ],
    CurrentVelocity := [ -39.37043543026334191381, -314.80982911633589083067, -743.63983854388607142027 ],
    CurrentAcceleration := [ 918.61171848468075040728, -8240.24070744882010330912, 376.40421615367449703626 ],
    TargetPosition := [ -38.32577323859909057546, 76.88839801585137934126, 77.24450399202348194194 ],
    TargetVelocity := [ 0.00000000000000000000, 0.00000000000000000000, 0.00000000000000000000 ],
    TargetAcceleration := [ 0.00000000000000000000, 0.00000000000000000000, 0.00000000000000000000 ]
  );
  
  positionExtrema : Struckig.PositionExtremaDesc;
END_VAR
TEST('Trajectory_32');

ruckig();

// Check total duration of profiles
AssertEquals_LREAL(Expected := 0.22561874467077386308, Actual := ruckig.Duration, DELTA := 1E-8, Message := 'Duration incorrect');

// Check duration for each phase
positionExtrema := ruckig._profiles[0].positionExtrema();
AssertEquals_LREAL(0.22561874467077389084, positionExtrema.Tmax, 1E-9, message:='Profile[0] Tmax incorrect');
AssertEquals_LREAL(-38.32577323859909057546, positionExtrema.Maximum, 1E-9, message:='Profile[0] maximum incorrect');
AssertEquals_LREAL(0.00883895720172546244, positionExtrema.Tmin, 1E-9, message:='Profile[0] Tmin incorrect');
AssertEquals_LREAL(-71.54075918203305661791, positionExtrema.Minimum, 1E-9, message:='Profile[0] minimum incorrect');

positionExtrema := ruckig._profiles[1].positionExtrema();
AssertEquals_LREAL(0.22561874448389260261, positionExtrema.Tmax, 1E-9, message:='Profile[1] Tmax incorrect');
AssertEquals_LREAL(76.88839801585137934126, positionExtrema.Maximum, 1E-9, message:='Profile[1] maximum incorrect');
AssertEquals_LREAL(0.04326693976782886031, positionExtrema.Tmin, 1E-9, message:='Profile[1] Tmin incorrect');
AssertEquals_LREAL(64.99037106700389188063, positionExtrema.Minimum, 1E-9, message:='Profile[1] minimum incorrect');

positionExtrema := ruckig._profiles[2].positionExtrema();
AssertEquals_LREAL(0.22561874467077386308, positionExtrema.Tmax, 1E-9, message:='Profile[2] Tmax incorrect');
AssertEquals_LREAL(77.24450399202348194194, positionExtrema.Maximum, 1E-9, message:='Profile[2] maximum incorrect');
AssertEquals_LREAL(0.02452949472980790746, positionExtrema.Tmin, 1E-9, message:='Profile[2] Tmin incorrect');
AssertEquals_LREAL(-47.33615887649365561174, positionExtrema.Minimum, 1E-9, message:='Profile[2] minimum incorrect');
   

TEST_FINISHED();
END_METHOD

METHOD Test_Trajectory_33
VAR_INST
  ruckig : Struckig.Ruckig(0.001, 3) := (
  
    Synchronization := SynchronizationType.TimeSync,        
    MaxVelocity := [ 2000.00000000000000000000, 2000.00000000000000000000, 2000.00000000000000000000 ],
    MaxAcceleration := [ 20000.00000000000000000000, 20000.00000000000000000000, 20000.00000000000000000000 ],
    MaxJerk := [ 800000.00000000000000000000, 800000.00000000000000000000, 800000.00000000000000000000 ],
    CurrentPosition := [ -10.72081173000827902797, -58.44147038088563306246, 98.86324493851924444243 ],
    CurrentVelocity := [ -408.47451658779903027607, -786.19958599415508615493, -998.10812621012325962511 ],
    CurrentAcceleration := [ 3503.92425371204808470793, 3035.68280271572984929662, -8529.36175578239635797217 ],
    TargetPosition := [ -24.74505052699171869790, -29.66847304289291287205, -86.07591857423138037575 ],
    TargetVelocity := [ 0.00000000000000000000, 0.00000000000000000000, 0.00000000000000000000 ],
    TargetAcceleration := [ 0.00000000000000000000, 0.00000000000000000000, 0.00000000000000000000 ]
  );
  
  positionExtrema : Struckig.PositionExtremaDesc;
END_VAR
TEST('Trajectory_33');

ruckig();

// Check total duration of profiles
AssertEquals_LREAL(Expected := 0.17123630970102474147, Actual := ruckig.Duration, DELTA := 1E-8, Message := 'Duration incorrect');

// Check duration for each phase
positionExtrema := ruckig._profiles[0].positionExtrema();
AssertEquals_LREAL(0.00000000000000000000, positionExtrema.Tmax, 1E-9, message:='Profile[0] Tmax incorrect');
AssertEquals_LREAL(-10.72081173000827902797, positionExtrema.Maximum, 1E-9, message:='Profile[0] maximum incorrect');
AssertEquals_LREAL(0.17123630970102476923, positionExtrema.Tmin, 1E-9, message:='Profile[0] Tmin incorrect');
AssertEquals_LREAL(-24.74505052699171869790, positionExtrema.Minimum, 1E-9, message:='Profile[0] minimum incorrect');

positionExtrema := ruckig._profiles[1].positionExtrema();
AssertEquals_LREAL(0.17123630970102471371, positionExtrema.Tmax, 1E-9, message:='Profile[1] Tmax incorrect');
AssertEquals_LREAL(-29.66847304289291287205, positionExtrema.Maximum, 1E-9, message:='Profile[1] maximum incorrect');
AssertEquals_LREAL(0.06908515615955748701, positionExtrema.Tmin, 1E-9, message:='Profile[1] Tmin incorrect');
AssertEquals_LREAL(-76.18339289032344652242, positionExtrema.Minimum, 1E-9, message:='Profile[1] minimum incorrect');

